LIN {X 0,Y 523.166,Z 946.333,A -85,B 0,C 180,E1 4773.992,E2 4773.992} C_VEL
LIN {X 0,Y 523.378,Z 938.631,A -85,B 0,C 180,E1 4777.898,E2 4777.898} C_VEL
LIN {X 0,Y 523.631,Z 926.038,A -85,B 0,C 180,E1 4781.677,E2 4781.677} C_VEL
LIN {X 0,Y 524.432,Z 907.467,A -85,B 0,C 180,E1 4785.488,E2 4785.488} C_VEL
LIN {X 0,Y 525.679,Z 882.892,A -85,B 0,C 180,E1 4789.124,E2 4789.124} C_VEL
LIN {X 0,Y 527.329,Z 854.452,A -85,B 0,C 180,E1 4792.218,E2 4792.218} C_VEL
LIN {X 0,Y 529.181,Z 823.204,A -85,B 0,C 180,E1 4794.735,E2 4794.735} C_VEL
LIN {X 0,Y 530.972,Z 787.135,A -85,B 0,C 180,E1 4796.792,E2 4796.792} C_VEL
LIN {X 0,Y 531.56,Z 762.454,A -85,B 0,C 180,E1 4797.793,E2 4797.793} C_VEL
LIN {X 0,Y 523.434,Z 741.053,A -85,B 0,C 180,E1 4799.156,E2 4799.156} C_VEL
LIN {X 0,Y 522.497,Z 737.44,A -85,B 0,C 180,E1 4799.385,E2 4799.385} C_VEL
LIN {X 0,Y 522.307,Z 737.44,A -85,B 0,C 180,E1 4805.432,E2 4805.432} C_VEL
LIN {X 0,Y 522.273,Z 737.44,A -85,B 0,C 180,E1 4811.816,E2 4811.816} C_VEL
LIN {X 0,Y 522.371,Z 737.44,A -85,B 0,C 180,E1 4818.204,E2 4818.204} C_VEL
LIN {X 0,Y 522.262,Z 737.44,A -85,B 0,C 180,E1 4824.573,E2 4824.573} C_VEL
LIN {X 0,Y 522.341,Z 737.44,A -85,B 0,C 180,E1 4830.487,E2 4830.487} C_VEL
LIN {X 0,Y 522.548,Z 737.44,A -85,B 0,C 180,E1 4836.077,E2 4836.077} C_VEL
LIN {X 0,Y 522.679,Z 737.44,A -85,B 0,C 180,E1 4841.426,E2 4841.426} C_VEL
LIN {X 0,Y 522.807,Z 737.44,A -85,B 0,C 180,E1 4846.61,E2 4846.61} C_VEL
LIN {X 0,Y 522.85,Z 737.44,A -85,B 0,C 180,E1 4851.68,E2 4851.68} C_VEL
LIN {X 0,Y 522.983,Z 737.44,A -85,B 0,C 180,E1 4856.685,E2 4856.685} C_VEL
LIN {X 0,Y 523.046,Z 737.44,A -85,B 0,C 180,E1 4861.663,E2 4861.663} C_VEL
LIN {X 0,Y 522.917,Z 737.44,A -85,B 0,C 180,E1 4866.654,E2 4866.654} C_VEL
LIN {X 0,Y 522.72,Z 737.44,A -85,B 0,C 180,E1 4871.701,E2 4871.701} C_VEL
LIN {X 0,Y 522.554,Z 737.44,A -85,B 0,C 180,E1 4877.039,E2 4877.039} C_VEL
LIN {X 0,Y 522.579,Z 737.44,A -85,B 0,C 180,E1 4882.128,E2 4882.128} C_VEL
LIN {X 0,Y 522.437,Z 737.44,A -85,B 0,C 180,E1 4887.627,E2 4887.627} C_VEL
LIN {X 0,Y 522.3,Z 737.44,A -85,B 0,C 180,E1 4892.5,E2 4892.5} C_VEL
LIN {X 0,Y 519.848,Z 737.44,A -85,B 0,C 180,E1 4893.914,E2 4893.914} C_VEL
LIN {X 0,Y 514.362,Z 737.44,A -85,B 0,C 180,E1 4896.278,E2 4896.278} C_VEL
LIN {X 0,Y 514.448,Z 737.44,A -85,B 0,C 180,E1 4900.351,E2 4900.351} C_VEL
LIN {X 0,Y 514.369,Z 737.44,A -85,B 0,C 180,E1 4905.056,E2 4905.056} C_VEL
LIN {X 0,Y 514.451,Z 738.219,A -85,B 0,C 180,E1 4908.773,E2 4908.773} C_VEL
LIN {X 0,Y 522.159,Z 752.872,A -85,B 0,C 180,E1 4909.551,E2 4909.551} C_VEL
LIN {X 0,Y 533.735,Z 774.419,A -85,B 0,C 180,E1 4910.952,E2 4910.952} C_VEL
LIN {X 0,Y 532.764,Z 835.83,A -85,B 0,C 180,E1 4912.111,E2 4912.111} C_VEL
LIN {X 0,Y 530.712,Z 877.373,A -85,B 0,C 180,E1 4913.563,E2 4913.563} C_VEL
LIN {X 0,Y 527.965,Z 915.757,A -85,B 0,C 180,E1 4915.56,E2 4915.56} C_VEL
LIN {X 0,Y 524.956,Z 952.662,A -85,B 0,C 180,E1 4918.186,E2 4918.186} C_VEL
LIN {X 0,Y 521.949,Z 987.101,A -85,B 0,C 180,E1 4921.405,E2 4921.405} C_VEL
LIN {X 0,Y 519.457,Z 1016.798,A -85,B 0,C 180,E1 4924.974,E2 4924.974} C_VEL
LIN {X 0,Y 517.473,Z 1044.169,A -85,B 0,C 180,E1 4929.222,E2 4929.222} C_VEL
LIN {X 0,Y 516.306,Z 1064.719,A -85,B 0,C 180,E1 4933.387,E2 4933.387} C_VEL
LIN {X 0,Y 515.508,Z 1081.773,A -85,B 0,C 180,E1 4938.136,E2 4938.136} C_VEL
LIN {X 0,Y 515.302,Z 1091.918,A -85,B 0,C 180,E1 4942.402,E2 4942.402} C_VEL
LIN {X 0,Y 515.21,Z 1097.627,A -85,B 0,C 180,E1 4946.631,E2 4946.631} C_VEL
LIN {X 0,Y 515.166,Z 1099,A -85,B 0,C 180,E1 4950,E2 4950} C_VEL
LIN {X 0,Y 515.206,Z 1097.628,A -85,B 0,C 180,E1 4953.369,E2 4953.369} C_VEL
LIN {X 0,Y 515.35,Z 1091.918,A -85,B 0,C 180,E1 4957.597,E2 4957.597} C_VEL
LIN {X 0,Y 515.5,Z 1081.775,A -85,B 0,C 180,E1 4961.864,E2 4961.864} C_VEL
LIN {X 0,Y 516.118,Z 1066.495,A -85,B 0,C 180,E1 4966.181,E2 4966.181} C_VEL
LIN {X 0,Y 517.333,Z 1045.386,A -85,B 0,C 180,E1 4970.56,E2 4970.56} C_VEL
LIN {X 0,Y 519.164,Z 1019.846,A -85,B 0,C 180,E1 4974.604,E2 4974.604} C_VEL
LIN {X 0,Y 521.782,Z 989.204,A -85,B 0,C 180,E1 4978.368,E2 4978.368} C_VEL
LIN {X 0,Y 524.709,Z 955.261,A -85,B 0,C 180,E1 4981.604,E2 4981.604} C_VEL
LIN {X 0,Y 527.867,Z 917.562,A -85,B 0,C 180,E1 4984.328,E2 4984.328} C_VEL
LIN {X 0,Y 530.645,Z 879.156,A -85,B 0,C 180,E1 4986.358,E2 4986.358} C_VEL
LIN {X 0,Y 532.759,Z 837.651,A -85,B 0,C 180,E1 4987.83,E2 4987.83} C_VEL
LIN {X 0,Y 533.918,Z 785.197,A -85,B 0,C 180,E1 4988.849,E2 4988.849} C_VEL
LIN {X 0,Y 533.297,Z 773.528,A -85,B 0,C 180,E1 4989.101,E2 4989.101} C_VEL
LIN {X 0,Y 515.632,Z 741.65,A -85,B 0,C 180,E1 4991.091,E2 4991.091} C_VEL
LIN {X 0,Y 514.405,Z 737.44,A -85,B 0,C 180,E1 4991.277,E2 4991.277} C_VEL
LIN {X 0,Y 514.421,Z 737.44,A -85,B 0,C 180,E1 4997.396,E2 4997.396} C_VEL
LIN {X 0,Y 514.375,Z 737.44,A -85,B 0,C 180,E1 5002.627,E2 5002.627} C_VEL
LIN {X 0,Y 514.427,Z 737.44,A -85,B 0,C 180,E1 5008.593,E2 5008.593} C_VEL
LIN {X 0,Y 514.57,Z 737.44,A -85,B 0,C 180,E1 5013.808,E2 5013.808} C_VEL
LIN {X 0,Y 514.7,Z 737.44,A -85,B 0,C 180,E1 5020.267,E2 5020.267} C_VEL
LIN {X 0,Y 514.536,Z 737.44,A -85,B 0,C 180,E1 5026.168,E2 5026.168} C_VEL
LIN {X 0,Y 514.81,Z 737.44,A -85,B 0,C 180,E1 5031.541,E2 5031.541} C_VEL
LIN {X 0,Y 514.936,Z 737.44,A -85,B 0,C 180,E1 5036.625,E2 5036.625} C_VEL
LIN {X 0,Y 514.939,Z 737.44,A -85,B 0,C 180,E1 5041.68,E2 5041.68} C_VEL
LIN {X 0,Y 514.889,Z 737.44,A -85,B 0,C 180,E1 5046.75,E2 5046.75} C_VEL
LIN {X 0,Y 514.767,Z 737.44,A -85,B 0,C 180,E1 5051.875,E2 5051.875} C_VEL
LIN {X 0,Y 514.697,Z 737.44,A -85,B 0,C 180,E1 5057.101,E2 5057.101} C_VEL
LIN {X 0,Y 514.616,Z 737.44,A -85,B 0,C 180,E1 5062.479,E2 5062.479} C_VEL
LIN {X 0,Y 514.462,Z 737.44,A -85,B 0,C 180,E1 5068.082,E2 5068.082} C_VEL
LIN {X 0,Y 514.395,Z 737.44,A -85,B 0,C 180,E1 5073.993,E2 5073.993} C_VEL
LIN {X 0,Y 514.349,Z 737.44,A -85,B 0,C 180,E1 5080.349,E2 5080.349} C_VEL
LIN {X 0,Y 514.405,Z 737.44,A -85,B 0,C 180,E1 5085.06,E2 5085.06} C_VEL
LIN {X 0,Y 514.451,Z 737.44,A -85,B 0,C 180,E1 5089.909,E2 5089.909} C_VEL
LIN {X 0,Y 514.344,Z 737.44,A -85,B 0,C 180,E1 5095.995,E2 5095.995} C_VEL
LIN {X 0,Y 514.356,Z 737.853,A -85,B 0,C 180,E1 5099.839,E2 5099.839} C_VEL
LIN {X 0,Y 523.372,Z 760.385,A -85,B 0,C 180,E1 5101.367,E2 5101.367} C_VEL
LIN {X 0,Y 525.202,Z 769.331,A -85,B 0,C 180,E1 5101.888,E2 5101.888} C_VEL
LIN {X 0,Y 523.014,Z 804.439,A -85,B 0,C 180,E1 5103.621,E2 5103.621} C_VEL
LIN {X 0,Y 520.977,Z 837.566,A -85,B 0,C 180,E1 5105.879,E2 5105.879} C_VEL
LIN {X 0,Y 518.918,Z 868.893,A -85,B 0,C 180,E1 5108.828,E2 5108.828} C_VEL
LIN {X 0,Y 517.233,Z 895.151,A -85,B 0,C 180,E1 5112.188,E2 5112.188} C_VEL
LIN {X 0,Y 516.175,Z 916.482,A -85,B 0,C 180,E1 5115.889,E2 5115.889} C_VEL
LIN {X 0,Y 515.578,Z 932.641,A -85,B 0,C 180,E1 5119.852,E2 5119.852} C_VEL
LIN {X 0,Y 515.345,Z 941.867,A -85,B 0,C 180,E1 5123.252,E2 5123.252} C_VEL
LIN {X 0,Y 515.228,Z 947.932,A -85,B 0,C 180,E1 5127.345,E2 5127.345} C_VEL
LIN {X 0,Y 515.27,Z 948.997,A -85,B 0,C 180,E1 5130,E2 5130} C_VEL
LIN {X 0,Y 515.281,Z 946.109,A -85,B 0,C 180,E1 5134.213,E2 5134.213} C_VEL
LIN {X 0,Y 515.507,Z 937.486,A -85,B 0,C 180,E1 5138.444,E2 5138.444} C_VEL
LIN {X 0,Y 515.887,Z 924.305,A -85,B 0,C 180,E1 5142.285,E2 5142.285} C_VEL
LIN {X 0,Y 516.782,Z 905.02,A -85,B 0,C 180,E1 5146.16,E2 5146.16} C_VEL
LIN {X 0,Y 518.157,Z 881.147,A -85,B 0,C 180,E1 5149.634,E2 5149.634} C_VEL
LIN {X 0,Y 519.898,Z 853.939,A -85,B 0,C 180,E1 5152.604,E2 5152.604} C_VEL
LIN {X 0,Y 522.023,Z 821.677,A -85,B 0,C 180,E1 5155.212,E2 5155.212} C_VEL
LIN {X 0,Y 524.446,Z 782.487,A -85,B 0,C 180,E1 5157.458,E2 5157.458} C_VEL
LIN {X 0,Y 524.782,Z 764.25,A -85,B 0,C 180,E1 5158.264,E2 5158.264} C_VEL
LIN {X 0,Y 516.75,Z 742.879,A -85,B 0,C 180,E1 5159.711,E2 5159.711} C_VEL
LIN {X 0,Y 514.477,Z 737.44,A -85,B 0,C 180,E1 5160.14,E2 5160.14} C_VEL
LIN {X 0,Y 514.374,Z 737.44,A -85,B 0,C 180,E1 5166.063,E2 5166.063} C_VEL
LIN {X 0,Y 514.361,Z 737.44,A -85,B 0,C 180,E1 5172.632,E2 5172.632} C_VEL
LIN {X 0,Y 514.44,Z 737.44,A -85,B 0,C 180,E1 5177.409,E2 5177.409} C_VEL
LIN {X 0,Y 514.388,Z 737.44,A -85,B 0,C 180,E1 5182.626,E2 5182.626} C_VEL
LIN {X 0,Y 514.391,Z 737.44,A -85,B 0,C 180,E1 5188.6,E2 5188.6} C_VEL
LIN {X 0,Y 514.568,Z 737.44,A -85,B 0,C 180,E1 5193.818,E2 5193.818} C_VEL
LIN {X 0,Y 514.745,Z 737.44,A -85,B 0,C 180,E1 5200.254,E2 5200.254} C_VEL
LIN {X 0,Y 514.878,Z 737.44,A -85,B 0,C 180,E1 5206.4,E2 5206.4} C_VEL
LIN {X 0,Y 514.96,Z 737.44,A -85,B 0,C 180,E1 5211.552,E2 5211.552} C_VEL
LIN {X 0,Y 515.072,Z 737.44,A -85,B 0,C 180,E1 5216.634,E2 5216.634} C_VEL
LIN {X 0,Y 515.079,Z 737.44,A -85,B 0,C 180,E1 5222.025,E2 5222.025} C_VEL
LIN {X 0,Y 515.005,Z 737.44,A -85,B 0,C 180,E1 5226.757,E2 5226.757} C_VEL
LIN {X 0,Y 514.79,Z 737.44,A -85,B 0,C 180,E1 5231.884,E2 5231.884} C_VEL
LIN {X 0,Y 514.657,Z 737.44,A -85,B 0,C 180,E1 5237.111,E2 5237.111} C_VEL
LIN {X 0,Y 514.634,Z 737.44,A -85,B 0,C 180,E1 5242.488,E2 5242.488} C_VEL
LIN {X 0,Y 514.487,Z 737.44,A -85,B 0,C 180,E1 5248.091,E2 5248.091} C_VEL
LIN {X 0,Y 514.35,Z 737.44,A -85,B 0,C 180,E1 5254.007,E2 5254.007} C_VEL
LIN {X 0,Y 514.362,Z 737.44,A -85,B 0,C 180,E1 5256.278,E2 5256.278} C_VEL
LIN {X 0,Y 513.06,Z 737.44,A -85,B 0,C 180,E1 5257.241,E2 5257.241} C_VEL
LIN {X 0,Y 506.448,Z 737.44,A -85,B 0,C 180,E1 5259.862,E2 5259.862} C_VEL
LIN {X 0,Y 506.359,Z 737.44,A -85,B 0,C 180,E1 5260.111,E2 5260.111} C_VEL
LIN {X 0,Y 506.386,Z 737.44,A -85,B 0,C 180,E1 5265.854,E2 5265.854} C_VEL
LIN {X 0,Y 506.497,Z 737.44,A -85,B 0,C 180,E1 5268.178,E2 5268.178} C_VEL
LIN {X 0,Y 513.949,Z 753.392,A -85,B 0,C 180,E1 5268.981,E2 5268.981} C_VEL
LIN {X 0,Y 527.557,Z 777.284,A -85,B 0,C 180,E1 5270.455,E2 5270.455} C_VEL
LIN {X 0,Y 526.518,Z 835.827,A -85,B 0,C 180,E1 5271.58,E2 5271.58} C_VEL
LIN {X 0,Y 524.251,Z 877.617,A -85,B 0,C 180,E1 5273.051,E2 5273.051} C_VEL
LIN {X 0,Y 521.225,Z 916.8,A -85,B 0,C 180,E1 5275.12,E2 5275.12} C_VEL
LIN {X 0,Y 517.926,Z 953.306,A -85,B 0,C 180,E1 5277.76,E2 5277.76} C_VEL
LIN {X 0,Y 514.769,Z 987.099,A -85,B 0,C 180,E1 5280.969,E2 5280.969} C_VEL
LIN {X 0,Y 511.911,Z 1018.16,A -85,B 0,C 180,E1 5284.777,E2 5284.777} C_VEL
LIN {X 0,Y 509.841,Z 1044.171,A -85,B 0,C 180,E1 5288.896,E2 5288.896} C_VEL
LIN {X 0,Y 508.557,Z 1064.718,A -85,B 0,C 180,E1 5293.126,E2 5293.126} C_VEL
LIN {X 0,Y 507.659,Z 1081.773,A -85,B 0,C 180,E1 5297.95,E2 5297.95} C_VEL
LIN {X 0,Y 507.404,Z 1091.918,A -85,B 0,C 180,E1 5302.283,E2 5302.283} C_VEL
LIN {X 0,Y 507.308,Z 1097.627,A -85,B 0,C 180,E1 5306.578,E2 5306.578} C_VEL
LIN {X 0,Y 507.281,Z 1099,A -85,B 0,C 180,E1 5310,E2 5310} C_VEL
LIN {X 0,Y 507.301,Z 1097.628,A -85,B 0,C 180,E1 5313.422,E2 5313.422} C_VEL
LIN {X 0,Y 507.443,Z 1091.919,A -85,B 0,C 180,E1 5317.716,E2 5317.716} C_VEL
LIN {X 0,Y 507.635,Z 1081.774,A -85,B 0,C 180,E1 5322.05,E2 5322.05} C_VEL
LIN {X 0,Y 508.325,Z 1066.496,A -85,B 0,C 180,E1 5326.436,E2 5326.436} C_VEL
LIN {X 0,Y 509.72,Z 1045.388,A -85,B 0,C 180,E1 5330.881,E2 5330.881} C_VEL
LIN {X 0,Y 511.755,Z 1019.261,A -85,B 0,C 180,E1 5335.07,E2 5335.07} C_VEL
LIN {X 0,Y 514.578,Z 989.203,A -85,B 0,C 180,E1 5338.802,E2 5338.802} C_VEL
LIN {X 0,Y 517.817,Z 954.813,A -85,B 0,C 180,E1 5342.114,E2 5342.114} C_VEL
LIN {X 0,Y 521.131,Z 918.687,A -85,B 0,C 180,E1 5344.76,E2 5344.76} C_VEL
LIN {X 0,Y 524.23,Z 878.854,A -85,B 0,C 180,E1 5346.891,E2 5346.891} C_VEL
LIN {X 0,Y 526.562,Z 837.056,A -85,B 0,C 180,E1 5348.376,E2 5348.376} C_VEL
LIN {X 0,Y 527.773,Z 780.555,A -85,B 0,C 180,E1 5349.469,E2 5349.469} C_VEL
LIN {X 0,Y 526.678,Z 775.495,A -85,B 0,C 180,E1 5349.655,E2 5349.655} C_VEL
LIN {X 0,Y 508.709,Z 743.577,A -85,B 0,C 180,E1 5351.557,E2 5351.557} C_VEL
LIN {X 0,Y 506.504,Z 737.44,A -85,B 0,C 180,E1 5351.882,E2 5351.882} C_VEL
LIN {X 0,Y 506.454,Z 737.44,A -85,B 0,C 180,E1 5358.361,E2 5358.361} C_VEL
LIN {X 0,Y 506.49,Z 737.44,A -85,B 0,C 180,E1 5363.811,E2 5363.811} C_VEL
LIN {X 0,Y 506.5,Z 737.44,A -85,B 0,C 180,E1 5370.094,E2 5370.094} C_VEL
LIN {X 0,Y 506.666,Z 737.44,A -85,B 0,C 180,E1 5375.267,E2 5375.267} C_VEL
LIN {X 0,Y 506.825,Z 737.44,A -85,B 0,C 180,E1 5380.814,E2 5380.814} C_VEL
LIN {X 0,Y 506.65,Z 737.44,A -85,B 0,C 180,E1 5386.166,E2 5386.166} C_VEL
LIN {X 0,Y 506.892,Z 737.44,A -85,B 0,C 180,E1 5391.407,E2 5391.407} C_VEL
LIN {X 0,Y 507.031,Z 737.44,A -85,B 0,C 180,E1 5396.572,E2 5396.572} C_VEL
LIN {X 0,Y 507.039,Z 737.44,A -85,B 0,C 180,E1 5401.706,E2 5401.706} C_VEL
LIN {X 0,Y 506.979,Z 737.44,A -85,B 0,C 180,E1 5406.855,E2 5406.855} C_VEL
LIN {X 0,Y 506.845,Z 737.44,A -85,B 0,C 180,E1 5412.064,E2 5412.064} C_VEL
LIN {X 0,Y 506.775,Z 737.44,A -85,B 0,C 180,E1 5417.376,E2 5417.376} C_VEL
LIN {X 0,Y 506.695,Z 737.44,A -85,B 0,C 180,E1 5422.85,E2 5422.85} C_VEL
LIN {X 0,Y 506.5,Z 737.44,A -85,B 0,C 180,E1 5428.564,E2 5428.564} C_VEL
LIN {X 0,Y 506.472,Z 737.44,A -85,B 0,C 180,E1 5434.6,E2 5434.6} C_VEL
LIN {X 0,Y 506.366,Z 737.44,A -85,B 0,C 180,E1 5441.121,E2 5441.121} C_VEL
LIN {X 0,Y 506.454,Z 737.44,A -85,B 0,C 180,E1 5446.563,E2 5446.563} C_VEL
LIN {X 0,Y 506.475,Z 737.44,A -85,B 0,C 180,E1 5453.284,E2 5453.284} C_VEL
LIN {X 0,Y 506.467,Z 737.589,A -85,B 0,C 180,E1 5459.073,E2 5459.073} C_VEL
LIN {X 0,Y 510.942,Z 747.555,A -85,B 0,C 180,E1 5459.778,E2 5459.778} C_VEL
LIN {X 0,Y 517.56,Z 764.656,A -85,B 0,C 180,E1 5461.014,E2 5461.014} C_VEL
LIN {X 0,Y 518.735,Z 773.411,A -85,B 0,C 180,E1 5461.501,E2 5461.501} C_VEL
LIN {X 0,Y 516.582,Z 805.176,A -85,B 0,C 180,E1 5463.115,E2 5463.115} C_VEL
LIN {X 0,Y 513.935,Z 835.367,A -85,B 0,C 180,E1 5465.295,E2 5465.295} C_VEL
LIN {X 0,Y 511.374,Z 869.182,A -85,B 0,C 180,E1 5468.535,E2 5468.535} C_VEL
LIN {X 0,Y 509.582,Z 895.145,A -85,B 0,C 180,E1 5471.912,E2 5471.912} C_VEL
LIN {X 0,Y 508.367,Z 916.884,A -85,B 0,C 180,E1 5475.75,E2 5475.75} C_VEL
LIN {X 0,Y 507.728,Z 932.639,A -85,B 0,C 180,E1 5479.694,E2 5479.694} C_VEL
LIN {X 0,Y 507.453,Z 941.866,A -85,B 0,C 180,E1 5483.146,E2 5483.146} C_VEL
LIN {X 0,Y 507.342,Z 947.212,A -85,B 0,C 180,E1 5486.578,E2 5486.578} C_VEL
LIN {X 0,Y 507.378,Z 948.997,A -85,B 0,C 180,E1 5490,E2 5490} C_VEL
LIN {X 0,Y 507.384,Z 946.111,A -85,B 0,C 180,E1 5494.278,E2 5494.278} C_VEL
LIN {X 0,Y 507.618,Z 937.488,A -85,B 0,C 180,E1 5498.576,E2 5498.576} C_VEL
LIN {X 0,Y 508.043,Z 924.308,A -85,B 0,C 180,E1 5502.477,E2 5502.477} C_VEL
LIN {X 0,Y 509.012,Z 905.023,A -85,B 0,C 180,E1 5506.413,E2 5506.413} C_VEL
LIN {X 0,Y 510.547,Z 881.152,A -85,B 0,C 180,E1 5509.939,E2 5509.939} C_VEL
LIN {X 0,Y 512.56,Z 852.585,A -85,B 0,C 180,E1 5513.082,E2 5513.082} C_VEL
LIN {X 0,Y 515.422,Z 818.696,A -85,B 0,C 180,E1 5515.909,E2 5515.909} C_VEL
LIN {X 0,Y 517.936,Z 786.373,A -85,B 0,C 180,E1 5517.826,E2 5517.826} C_VEL
LIN {X 0,Y 518.495,Z 767.008,A -85,B 0,C 180,E1 5518.714,E2 5518.714} C_VEL
LIN {X 0,Y 511.71,Z 748.352,A -85,B 0,C 180,E1 5520.036,E2 5520.036} C_VEL
LIN {X 0,Y 506.639,Z 738.499,A -85,B 0,C 180,E1 5520.799,E2 5520.799} C_VEL
LIN {X 0,Y 506.562,Z 737.44,A -85,B 0,C 180,E1 5520.896,E2 5520.896} C_VEL
LIN {X 0,Y 506.44,Z 737.44,A -85,B 0,C 180,E1 5526.719,E2 5526.719} C_VEL
LIN {X 0,Y 506.401,Z 737.44,A -85,B 0,C 180,E1 5533.443,E2 5533.443} C_VEL
LIN {X 0,Y 506.445,Z 737.44,A -85,B 0,C 180,E1 5538.887,E2 5538.887} C_VEL
LIN {X 0,Y 506.42,Z 737.44,A -85,B 0,C 180,E1 5545.396,E2 5545.396} C_VEL
LIN {X 0,Y 506.496,Z 737.44,A -85,B 0,C 180,E1 5551.436,E2 5551.436} C_VEL
LIN {X 0,Y 506.707,Z 737.44,A -85,B 0,C 180,E1 5557.15,E2 5557.15} C_VEL
LIN {X 0,Y 506.904,Z 737.44,A -85,B 0,C 180,E1 5562.893,E2 5562.893} C_VEL
LIN {X 0,Y 506.918,Z 737.44,A -85,B 0,C 180,E1 5567.938,E2 5567.938} C_VEL
LIN {X 0,Y 506.982,Z 737.44,A -85,B 0,C 180,E1 5573.145,E2 5573.145} C_VEL
LIN {X 0,Y 507.041,Z 737.44,A -85,B 0,C 180,E1 5578.294,E2 5578.294} C_VEL
LIN {X 0,Y 507.033,Z 737.44,A -85,B 0,C 180,E1 5583.428,E2 5583.428} C_VEL
LIN {X 0,Y 506.906,Z 737.44,A -85,B 0,C 180,E1 5588.592,E2 5588.592} C_VEL
LIN {X 0,Y 506.821,Z 737.44,A -85,B 0,C 180,E1 5593.83,E2 5593.83} C_VEL
LIN {X 0,Y 506.7,Z 737.44,A -85,B 0,C 180,E1 5599.191,E2 5599.191} C_VEL
LIN {X 0,Y 506.668,Z 737.44,A -85,B 0,C 180,E1 5604.732,E2 5604.732} C_VEL
LIN {X 0,Y 506.489,Z 737.44,A -85,B 0,C 180,E1 5610.544,E2 5610.544} C_VEL
LIN {X 0,Y 506.473,Z 737.44,A -85,B 0,C 180,E1 5616.719,E2 5616.719} C_VEL
LIN {X 0,Y 506.359,Z 737.44,A -85,B 0,C 180,E1 5620.111,E2 5620.111} C_VEL
LIN {X 0,Y 503.864,Z 737.44,A -85,B 0,C 180,E1 5621.571,E2 5621.571} C_VEL
LIN {X 0,Y 498.587,Z 737.44,A -85,B 0,C 180,E1 5623.761,E2 5623.761} C_VEL
LIN {X 0,Y 498.5,Z 737.44,A -85,B 0,C 180,E1 5624.014,E2 5624.014} C_VEL
LIN {X 0,Y 498.611,Z 737.44,A -85,B 0,C 180,E1 5627.574,E2 5627.574} C_VEL
LIN {X 0,Y 508.319,Z 758.234,A -85,B 0,C 180,E1 5628.658,E2 5628.658} C_VEL
LIN {X 0,Y 521.561,Z 781.726,A -85,B 0,C 180,E1 5629.988,E2 5629.988} C_VEL
LIN {X 0,Y 520.326,Z 835.779,A -85,B 0,C 180,E1 5631.035,E2 5631.035} C_VEL
LIN {X 0,Y 517.807,Z 878.549,A -85,B 0,C 180,E1 5632.558,E2 5632.558} C_VEL
LIN {X 0,Y 514.461,Z 918.701,A -85,B 0,C 180,E1 5634.723,E2 5634.723} C_VEL
LIN {X 0,Y 510.665,Z 957.552,A -85,B 0,C 180,E1 5637.631,E2 5637.631} C_VEL
LIN {X 0,Y 506.956,Z 993.552,A -85,B 0,C 180,E1 5641.231,E2 5641.231} C_VEL
LIN {X 0,Y 503.768,Z 1025.525,A -85,B 0,C 180,E1 5645.45,E2 5645.45} C_VEL
LIN {X 0,Y 501.524,Z 1051.369,A -85,B 0,C 180,E1 5649.928,E2 5649.928} C_VEL
LIN {X 0,Y 500.246,Z 1071.518,A -85,B 0,C 180,E1 5654.596,E2 5654.596} C_VEL
LIN {X 0,Y 499.635,Z 1085.29,A -85,B 0,C 180,E1 5659.083,E2 5659.083} C_VEL
LIN {X 0,Y 499.476,Z 1093.479,A -85,B 0,C 180,E1 5663.036,E2 5663.036} C_VEL
LIN {X 0,Y 499.406,Z 1097.627,A -85,B 0,C 180,E1 5666.524,E2 5666.524} C_VEL
LIN {X 0,Y 499.4,Z 1099,A -85,B 0,C 180,E1 5670,E2 5670} C_VEL
LIN {X 0,Y 499.395,Z 1097.628,A -85,B 0,C 180,E1 5673.476,E2 5673.476} C_VEL
LIN {X 0,Y 499.553,Z 1091.919,A -85,B 0,C 180,E1 5677.838,E2 5677.838} C_VEL
LIN {X 0,Y 499.772,Z 1081.774,A -85,B 0,C 180,E1 5682.243,E2 5682.243} C_VEL
LIN {X 0,Y 500.551,Z 1066.497,A -85,B 0,C 180,E1 5686.699,E2 5686.699} C_VEL
LIN {X 0,Y 502.07,Z 1045.389,A -85,B 0,C 180,E1 5691.214,E2 5691.214} C_VEL
LIN {X 0,Y 504.311,Z 1018.984,A -85,B 0,C 180,E1 5695.507,E2 5695.507} C_VEL
LIN {X 0,Y 507.328,Z 989.675,A -85,B 0,C 180,E1 5699.198,E2 5699.198} C_VEL
LIN {X 0,Y 510.781,Z 956.306,A -85,B 0,C 180,E1 5702.475,E2 5702.475} C_VEL
LIN {X 0,Y 514.484,Z 918.702,A -85,B 0,C 180,E1 5705.275,E2 5705.275} C_VEL
LIN {X 0,Y 517.833,Z 879.033,A -85,B 0,C 180,E1 5707.415,E2 5707.415} C_VEL
LIN {X 0,Y 520.32,Z 837.566,A -85,B 0,C 180,E1 5708.905,E2 5708.905} C_VEL
LIN {X 0,Y 521.655,Z 784.779,A -85,B 0,C 180,E1 5709.95,E2 5709.95} C_VEL
LIN {X 0,Y 520.604,Z 778.711,A -85,B 0,C 180,E1 5710.144,E2 5710.144} C_VEL
LIN {X 0,Y 501.405,Z 744.954,A -85,B 0,C 180,E1 5712.079,E2 5712.079} C_VEL
LIN {X 0,Y 498.583,Z 737.44,A -85,B 0,C 180,E1 5712.484,E2 5712.484} C_VEL
LIN {X 0,Y 498.52,Z 737.44,A -85,B 0,C 180,E1 5718.075,E2 5718.075} C_VEL
LIN {X 0,Y 498.527,Z 737.44,A -85,B 0,C 180,E1 5724.757,E2 5724.757} C_VEL
LIN {X 0,Y 498.579,Z 737.44,A -85,B 0,C 180,E1 5730.929,E2 5730.929} C_VEL
LIN {X 0,Y 498.765,Z 737.44,A -85,B 0,C 180,E1 5736.755,E2 5736.755} C_VEL
LIN {X 0,Y 498.881,Z 737.44,A -85,B 0,C 180,E1 5742.33,E2 5742.33} C_VEL
LIN {X 0,Y 498.808,Z 737.44,A -85,B 0,C 180,E1 5747.73,E2 5747.73} C_VEL
LIN {X 0,Y 499.158,Z 737.44,A -85,B 0,C 180,E1 5753.028,E2 5753.028} C_VEL
LIN {X 0,Y 499.381,Z 737.44,A -85,B 0,C 180,E1 5758.258,E2 5758.258} C_VEL
LIN {X 0,Y 499.273,Z 737.44,A -85,B 0,C 180,E1 5763.472,E2 5763.472} C_VEL
LIN {X 0,Y 499.102,Z 737.44,A -85,B 0,C 180,E1 5768.718,E2 5768.718} C_VEL
LIN {X 0,Y 498.934,Z 737.44,A -85,B 0,C 180,E1 5774.043,E2 5774.043} C_VEL
LIN {X 0,Y 498.8,Z 737.44,A -85,B 0,C 180,E1 5779.792,E2 5779.792} C_VEL
LIN {X 0,Y 498.7,Z 737.44,A -85,B 0,C 180,E1 5785.145,E2 5785.145} C_VEL
LIN {X 0,Y 498.542,Z 737.44,A -85,B 0,C 180,E1 5791.755,E2 5791.755} C_VEL
LIN {X 0,Y 498.427,Z 737.44,A -85,B 0,C 180,E1 5797.837,E2 5797.837} C_VEL
LIN {X 0,Y 498.517,Z 737.44,A -85,B 0,C 180,E1 5804.296,E2 5804.296} C_VEL
LIN {X 0,Y 498.485,Z 737.44,A -85,B 0,C 180,E1 5810.372,E2 5810.372} C_VEL
LIN {X 0,Y 498.521,Z 737.44,A -85,B 0,C 180,E1 5816.862,E2 5816.862} C_VEL
LIN {X 0,Y 498.562,Z 737.44,A -85,B 0,C 180,E1 5818.257,E2 5818.257} C_VEL
LIN {X 0,Y 503.137,Z 747.617,A -85,B 0,C 180,E1 5819.011,E2 5819.011} C_VEL
LIN {X 0,Y 510.321,Z 763.929,A -85,B 0,C 180,E1 5820.297,E2 5820.297} C_VEL
LIN {X 0,Y 512.504,Z 774.93,A -85,B 0,C 180,E1 5820.992,E2 5820.992} C_VEL
LIN {X 0,Y 510.118,Z 807.352,A -85,B 0,C 180,E1 5822.673,E2 5822.673} C_VEL
LIN {X 0,Y 507.149,Z 837.974,A -85,B 0,C 180,E1 5824.942,E2 5824.942} C_VEL
LIN {X 0,Y 504.062,Z 868.129,A -85,B 0,C 180,E1 5828.041,E2 5828.041} C_VEL
LIN {X 0,Y 501.844,Z 896.264,A -85,B 0,C 180,E1 5831.798,E2 5831.798} C_VEL
LIN {X 0,Y 500.507,Z 918.03,A -85,B 0,C 180,E1 5835.769,E2 5835.769} C_VEL
LIN {X 0,Y 499.856,Z 932.637,A -85,B 0,C 180,E1 5839.53,E2 5839.53} C_VEL
LIN {X 0,Y 499.561,Z 941.865,A -85,B 0,C 180,E1 5843.037,E2 5843.037} C_VEL
LIN {X 0,Y 499.471,Z 947.211,A -85,B 0,C 180,E1 5846.525,E2 5846.525} C_VEL
LIN {X 0,Y 499.498,Z 948.997,A -85,B 0,C 180,E1 5850,E2 5850} C_VEL
LIN {X 0,Y 499.501,Z 946.111,A -85,B 0,C 180,E1 5854.346,E2 5854.346} C_VEL
LIN {X 0,Y 499.764,Z 937.49,A -85,B 0,C 180,E1 5858.712,E2 5858.712} C_VEL
LIN {X 0,Y 500.218,Z 924.31,A -85,B 0,C 180,E1 5862.676,E2 5862.676} C_VEL
LIN {X 0,Y 501.28,Z 905.026,A -85,B 0,C 180,E1 5866.674,E2 5866.674} C_VEL
LIN {X 0,Y 502.948,Z 881.157,A -85,B 0,C 180,E1 5870.254,E2 5870.254} C_VEL
LIN {X 0,Y 505.934,Z 849.575,A -85,B 0,C 180,E1 5873.896,E2 5873.896} C_VEL
LIN {X 0,Y 508.912,Z 820.136,A -85,B 0,C 180,E1 5876.384,E2 5876.384} C_VEL
LIN {X 0,Y 511.63,Z 787.99,A -85,B 0,C 180,E1 5878.322,E2 5878.322} C_VEL
LIN {X 0,Y 512.161,Z 769.312,A -85,B 0,C 180,E1 5879.211,E2 5879.211} C_VEL
LIN {X 0,Y 505.862,Z 752.546,A -85,B 0,C 180,E1 5880.469,E2 5880.469} C_VEL
LIN {X 0,Y 498.805,Z 739.066,A -85,B 0,C 180,E1 5881.575,E2 5881.575} C_VEL
LIN {X 0,Y 498.635,Z 737.44,A -85,B 0,C 180,E1 5881.718,E2 5881.718} C_VEL
LIN {X 0,Y 498.425,Z 737.44,A -85,B 0,C 180,E1 5887.85,E2 5887.85} C_VEL
LIN {X 0,Y 498.505,Z 737.44,A -85,B 0,C 180,E1 5894.309,E2 5894.309} C_VEL
LIN {X 0,Y 498.48,Z 737.44,A -85,B 0,C 180,E1 5900.381,E2 5900.381} C_VEL
LIN {X 0,Y 498.484,Z 737.44,A -85,B 0,C 180,E1 5906.868,E2 5906.868} C_VEL
LIN {X 0,Y 498.627,Z 737.44,A -85,B 0,C 180,E1 5912.914,E2 5912.914} C_VEL
LIN {X 0,Y 498.846,Z 737.44,A -85,B 0,C 180,E1 5918.648,E2 5918.648} C_VEL
LIN {X 0,Y 498.986,Z 737.44,A -85,B 0,C 180,E1 5924.159,E2 5924.159} C_VEL
LIN {X 0,Y 499.093,Z 737.44,A -85,B 0,C 180,E1 5929.519,E2 5929.519} C_VEL
LIN {X 0,Y 499.141,Z 737.44,A -85,B 0,C 180,E1 5934.784,E2 5934.784} C_VEL
LIN {X 0,Y 499.255,Z 737.44,A -85,B 0,C 180,E1 5940.005,E2 5940.005} C_VEL
LIN {X 0,Y 499.165,Z 737.44,A -85,B 0,C 180,E1 5945.225,E2 5945.225} C_VEL
LIN {X 0,Y 499.003,Z 737.44,A -85,B 0,C 180,E1 5950.492,E2 5950.492} C_VEL
LIN {X 0,Y 498.86,Z 737.44,A -85,B 0,C 180,E1 5955.855,E2 5955.855} C_VEL
LIN {X 0,Y 498.792,Z 737.44,A -85,B 0,C 180,E1 5961.364,E2 5961.364} C_VEL
LIN {X 0,Y 498.64,Z 737.44,A -85,B 0,C 180,E1 5967.096,E2 5967.096} C_VEL
LIN {X 0,Y 498.502,Z 737.44,A -85,B 0,C 180,E1 5973.141,E2 5973.141} C_VEL
LIN {X 0,Y 498.486,Z 737.44,A -85,B 0,C 180,E1 5979.631,E2 5979.631} C_VEL
LIN {X 0,Y 498.5,Z 737.44,A -85,B 0,C 180,E1 5984.014,E2 5984.014} C_VEL
LIN {X 0,Y 494.524,Z 737.44,A -85,B 0,C 180,E1 5985.297,E2 5985.297} C_VEL
LIN {X 0,Y 490.596,Z 737.44,A -85,B 0,C 180,E1 5986.601,E2 5986.601} C_VEL
LIN {X 0,Y 490.662,Z 738.171,A -85,B 0,C 180,E1 5986.978,E2 5986.978} C_VEL
LIN {X 0,Y 504.962,Z 766.638,A -85,B 0,C 180,E1 5988.553,E2 5988.553} C_VEL
LIN {X 0,Y 514.956,Z 784.586,A -85,B 0,C 180,E1 5989.552,E2 5989.552} C_VEL
LIN {X 0,Y 513.998,Z 837.096,A -85,B 0,C 180,E1 5990.533,E2 5990.533} C_VEL
LIN {X 0,Y 511.554,Z 877.526,A -85,B 0,C 180,E1 5991.969,E2 5991.969} C_VEL
LIN {X 0,Y 507.881,Z 918.693,A -85,B 0,C 180,E1 5994.196,E2 5994.196} C_VEL
LIN {X 0,Y 503.793,Z 957.498,A -85,B 0,C 180,E1 5997.129,E2 5997.129} C_VEL
LIN {X 0,Y 499.776,Z 993.772,A -85,B 0,C 180,E1 6000.805,E2 6000.805} C_VEL
LIN {X 0,Y 496.373,Z 1024.941,A -85,B 0,C 180,E1 6004.963,E2 6004.963} C_VEL
LIN {X 0,Y 493.982,Z 1050.272,A -85,B 0,C 180,E1 6009.377,E2 6009.377} C_VEL
LIN {X 0,Y 492.575,Z 1069.983,A -85,B 0,C 180,E1 6013.941,E2 6013.941} C_VEL
LIN {X 0,Y 491.834,Z 1084.143,A -85,B 0,C 180,E1 6018.458,E2 6018.458} C_VEL
LIN {X 0,Y 491.579,Z 1093.479,A -85,B 0,C 180,E1 6022.923,E2 6022.923} C_VEL
LIN {X 0,Y 491.504,Z 1097.627,A -85,B 0,C 180,E1 6026.468,E2 6026.468} C_VEL
LIN {X 0,Y 491.5,Z 1099,A -85,B 0,C 180,E1 6030,E2 6030} C_VEL
LIN {X 0,Y 491.49,Z 1097.628,A -85,B 0,C 180,E1 6033.532,E2 6033.532} C_VEL
LIN {X 0,Y 491.655,Z 1091.919,A -85,B 0,C 180,E1 6037.965,E2 6037.965} C_VEL
LIN {X 0,Y 491.92,Z 1081.773,A -85,B 0,C 180,E1 6042.441,E2 6042.441} C_VEL
LIN {X 0,Y 492.908,Z 1064.858,A -85,B 0,C 180,E1 6047.391,E2 6047.391} C_VEL
LIN {X 0,Y 494.728,Z 1041.691,A -85,B 0,C 180,E1 6052.253,E2 6052.253} C_VEL
LIN {X 0,Y 497.557,Z 1013.532,A -85,B 0,C 180,E1 6056.688,E2 6056.688} C_VEL
LIN {X 0,Y 501.095,Z 981.672,A -85,B 0,C 180,E1 6060.539,E2 6060.539} C_VEL
LIN {X 0,Y 505.114,Z 945.518,A -85,B 0,C 180,E1 6063.876,E2 6063.876} C_VEL
LIN {X 0,Y 509.08,Z 905.991,A -85,B 0,C 180,E1 6066.584,E2 6066.584} C_VEL
LIN {X 0,Y 512.617,Z 863.483,A -85,B 0,C 180,E1 6068.61,E2 6068.61} C_VEL
LIN {X 0,Y 514.701,Z 824.962,A -85,B 0,C 180,E1 6069.737,E2 6069.737} C_VEL
LIN {X 0,Y 514.432,Z 782.453,A -85,B 0,C 180,E1 6070.517,E2 6070.517} C_VEL
LIN {X 0,Y 495.559,Z 749.173,A -85,B 0,C 180,E1 6072.45,E2 6072.45} C_VEL
LIN {X 0,Y 490.657,Z 737.44,A -85,B 0,C 180,E1 6073.086,E2 6073.086} C_VEL
LIN {X 0,Y 490.561,Z 737.44,A -85,B 0,C 180,E1 6079.599,E2 6079.599} C_VEL
LIN {X 0,Y 490.583,Z 737.44,A -85,B 0,C 180,E1 6086.253,E2 6086.253} C_VEL
LIN {X 0,Y 490.695,Z 737.44,A -85,B 0,C 180,E1 6092.429,E2 6092.429} C_VEL
LIN {X 0,Y 490.87,Z 737.44,A -85,B 0,C 180,E1 6098.274,E2 6098.274} C_VEL
LIN {X 0,Y 490.889,Z 737.44,A -85,B 0,C 180,E1 6103.881,E2 6103.881} C_VEL
LIN {X 0,Y 491.021,Z 737.44,A -85,B 0,C 180,E1 6110.634,E2 6110.634} C_VEL
LIN {X 0,Y 491.222,Z 737.44,A -85,B 0,C 180,E1 6116.462,E2 6116.462} C_VEL
LIN {X 0,Y 491.252,Z 737.44,A -85,B 0,C 180,E1 6121.761,E2 6121.761} C_VEL
LIN {X 0,Y 491.156,Z 737.44,A -85,B 0,C 180,E1 6127.077,E2 6127.077} C_VEL
LIN {X 0,Y 491.013,Z 737.44,A -85,B 0,C 180,E1 6132.459,E2 6132.459} C_VEL
LIN {X 0,Y 490.922,Z 737.44,A -85,B 0,C 180,E1 6137.956,E2 6137.956} C_VEL
LIN {X 0,Y 490.807,Z 737.44,A -85,B 0,C 180,E1 6143.634,E2 6143.634} C_VEL
LIN {X 0,Y 490.603,Z 737.44,A -85,B 0,C 180,E1 6150.223,E2 6150.223} C_VEL
LIN {X 0,Y 490.543,Z 737.44,A -85,B 0,C 180,E1 6155.893,E2 6155.893} C_VEL
LIN {X 0,Y 490.59,Z 737.44,A -85,B 0,C 180,E1 6162.75,E2 6162.75} C_VEL
LIN {X 0,Y 490.634,Z 737.44,A -85,B 0,C 180,E1 6167.769,E2 6167.769} C_VEL
LIN {X 0,Y 490.546,Z 737.44,A -85,B 0,C 180,E1 6174.098,E2 6174.098} C_VEL
LIN {X 0,Y 490.609,Z 737.44,A -85,B 0,C 180,E1 6177.439,E2 6177.439} C_VEL
LIN {X 0,Y 495.098,Z 747.292,A -85,B 0,C 180,E1 6178.17,E2 6178.17} C_VEL
LIN {X 0,Y 504.455,Z 767.587,A -85,B 0,C 180,E1 6179.869,E2 6179.869} C_VEL
LIN {X 0,Y 506.306,Z 777.052,A -85,B 0,C 180,E1 6180.491,E2 6180.491} C_VEL
LIN {X 0,Y 503.681,Z 809.848,A -85,B 0,C 180,E1 6182.232,E2 6182.232} C_VEL
LIN {X 0,Y 500.412,Z 840.69,A -85,B 0,C 180,E1 6184.581,E2 6184.581} C_VEL
LIN {X 0,Y 497.146,Z 869.582,A -85,B 0,C 180,E1 6187.625,E2 6187.625} C_VEL
LIN {X 0,Y 494.337,Z 894.601,A -85,B 0,C 180,E1 6191.222,E2 6191.222} C_VEL
LIN {X 0,Y 492.862,Z 916.201,A -85,B 0,C 180,E1 6195.15,E2 6195.15} C_VEL
LIN {X 0,Y 491.997,Z 932.635,A -85,B 0,C 180,E1 6199.36,E2 6199.36} C_VEL
LIN {X 0,Y 491.671,Z 941.863,A -85,B 0,C 180,E1 6202.925,E2 6202.925} C_VEL
LIN {X 0,Y 491.57,Z 947.21,A -85,B 0,C 180,E1 6206.469,E2 6206.469} C_VEL
LIN {X 0,Y 491.598,Z 948.997,A -85,B 0,C 180,E1 6210,E2 6210} C_VEL
LIN {X 0,Y 491.621,Z 946.112,A -85,B 0,C 180,E1 6214.416,E2 6214.416} C_VEL
LIN {X 0,Y 491.872,Z 937.492,A -85,B 0,C 180,E1 6218.853,E2 6218.853} C_VEL
LIN {X 0,Y 492.393,Z 924.312,A -85,B 0,C 180,E1 6222.881,E2 6222.881} C_VEL
LIN {X 0,Y 493.512,Z 905.029,A -85,B 0,C 180,E1 6226.944,E2 6226.944} C_VEL
LIN {X 0,Y 496.354,Z 875.948,A -85,B 0,C 180,E1 6231.471,E2 6231.471} C_VEL
LIN {X 0,Y 499.539,Z 848.228,A -85,B 0,C 180,E1 6234.622,E2 6234.622} C_VEL
LIN {X 0,Y 502.796,Z 818.54,A -85,B 0,C 180,E1 6237.095,E2 6237.095} C_VEL
LIN {X 0,Y 505.654,Z 786.108,A -85,B 0,C 180,E1 6239.011,E2 6239.011} C_VEL
LIN {X 0,Y 506.208,Z 772.998,A -85,B 0,C 180,E1 6239.629,E2 6239.629} C_VEL
LIN {X 0,Y 500.555,Z 757.483,A -85,B 0,C 180,E1 6240.837,E2 6240.837} C_VEL
LIN {X 0,Y 490.939,Z 739.339,A -85,B 0,C 180,E1 6242.364,E2 6242.364} C_VEL
LIN {X 0,Y 490.684,Z 737.44,A -85,B 0,C 180,E1 6242.521,E2 6242.521} C_VEL
LIN {X 0,Y 490.494,Z 737.44,A -85,B 0,C 180,E1 6248.122,E2 6248.122} C_VEL
LIN {X 0,Y 490.583,Z 737.44,A -85,B 0,C 180,E1 6252.761,E2 6252.761} C_VEL
LIN {X 0,Y 490.637,Z 737.44,A -85,B 0,C 180,E1 6257.781,E2 6257.781} C_VEL
LIN {X 0,Y 490.52,Z 737.44,A -85,B 0,C 180,E1 6264.105,E2 6264.105} C_VEL
LIN {X 0,Y 490.588,Z 737.44,A -85,B 0,C 180,E1 6270.419,E2 6270.419} C_VEL
LIN {X 0,Y 490.824,Z 737.44,A -85,B 0,C 180,E1 6276.367,E2 6276.367} C_VEL
LIN {X 0,Y 490.997,Z 737.44,A -85,B 0,C 180,E1 6282.047,E2 6282.047} C_VEL
LIN {X 0,Y 491.09,Z 737.44,A -85,B 0,C 180,E1 6287.543,E2 6287.543} C_VEL
LIN {X 0,Y 491.164,Z 737.44,A -85,B 0,C 180,E1 6292.923,E2 6292.923} C_VEL
LIN {X 0,Y 491.254,Z 737.44,A -85,B 0,C 180,E1 6298.239,E2 6298.239} C_VEL
LIN {X 0,Y 491.224,Z 737.44,A -85,B 0,C 180,E1 6303.538,E2 6303.538} C_VEL
LIN {X 0,Y 491.054,Z 737.44,A -85,B 0,C 180,E1 6309.388,E2 6309.388} C_VEL
LIN {X 0,Y 490.967,Z 737.44,A -85,B 0,C 180,E1 6314.286,E2 6314.286} C_VEL
LIN {X 0,Y 490.854,Z 737.44,A -85,B 0,C 180,E1 6319.836,E2 6319.836} C_VEL
LIN {X 0,Y 490.771,Z 737.44,A -85,B 0,C 180,E1 6325.59,E2 6325.59} C_VEL
LIN {X 0,Y 490.609,Z 737.44,A -85,B 0,C 180,E1 6331.644,E2 6331.644} C_VEL
LIN {X 0,Y 490.555,Z 737.44,A -85,B 0,C 180,E1 6338.118,E2 6338.118} C_VEL
LIN {X 0,Y 490.536,Z 737.44,A -85,B 0,C 180,E1 6344.016,E2 6344.016} C_VEL
LIN {X 0,Y 490.596,Z 737.44,A -85,B 0,C 180,E1 6346.601,E2 6346.601} C_VEL
LIN {X 0,Y 492.101,Z 740.218,A -85,B 0,C 180,E1 6347.102,E2 6347.102} C_VEL
LIN {X 0,Y 494.637,Z 749.813,A -85,B 0,C 180,E1 6347.496,E2 6347.496} C_VEL
LIN {X 0,Y 496.996,Z 767.013,A -85,B 0,C 180,E1 6347.975,E2 6347.975} C_VEL
LIN {X 0,Y 497.957,Z 769.12,A -85,B 0,C 180,E1 6348.087,E2 6348.087} C_VEL
LIN {X 0,Y 508.222,Z 786.689,A -85,B 0,C 180,E1 6349.118,E2 6349.118} C_VEL
LIN {X 0,Y 507.118,Z 838.063,A -85,B 0,C 180,E1 6350.113,E2 6350.113} C_VEL
LIN {X 0,Y 504.832,Z 880.073,A -85,B 0,C 180,E1 6351.561,E2 6351.561} C_VEL
LIN {X 0,Y 501.474,Z 917.434,A -85,B 0,C 180,E1 6353.577,E2 6353.577} C_VEL
LIN {X 0,Y 497.064,Z 956.239,A -85,B 0,C 180,E1 6356.507,E2 6356.507} C_VEL
LIN {X 0,Y 492.934,Z 990.85,A -85,B 0,C 180,E1 6360.005,E2 6360.005} C_VEL
LIN {X 0,Y 489.252,Z 1022.003,A -85,B 0,C 180,E1 6364.115,E2 6364.115} C_VEL
LIN {X 0,Y 486.589,Z 1048.238,A -85,B 0,C 180,E1 6368.645,E2 6368.645} C_VEL
LIN {X 0,Y 484.971,Z 1068.384,A -85,B 0,C 180,E1 6373.253,E2 6373.253} C_VEL
LIN {X 0,Y 484.063,Z 1082.989,A -85,B 0,C 180,E1 6377.812,E2 6377.812} C_VEL
LIN {X 0,Y 483.7,Z 1093.479,A -85,B 0,C 180,E1 6382.808,E2 6382.808} C_VEL
LIN {X 0,Y 483.608,Z 1097.627,A -85,B 0,C 180,E1 6386.41,E2 6386.41} C_VEL
LIN {X 0,Y 483.63,Z 1099,A -85,B 0,C 180,E1 6390,E2 6390} C_VEL
LIN {X 0,Y 483.595,Z 1097.628,A -85,B 0,C 180,E1 6393.59,E2 6393.59} C_VEL
LIN {X 0,Y 483.776,Z 1091.919,A -85,B 0,C 180,E1 6398.096,E2 6398.096} C_VEL
LIN {X 0,Y 484.063,Z 1081.773,A -85,B 0,C 180,E1 6402.646,E2 6402.646} C_VEL
LIN {X 0,Y 485.15,Z 1064.909,A -85,B 0,C 180,E1 6407.666,E2 6407.666} C_VEL
LIN {X 0,Y 487.206,Z 1041.715,A -85,B 0,C 180,E1 6412.611,E2 6412.611} C_VEL
LIN {X 0,Y 490.136,Z 1014.345,A -85,B 0,C 180,E1 6417.01,E2 6417.01} C_VEL
LIN {X 0,Y 494.064,Z 981.716,A -85,B 0,C 180,E1 6421.017,E2 6421.017} C_VEL
LIN {X 0,Y 498.483,Z 944.625,A -85,B 0,C 180,E1 6424.466,E2 6424.466} C_VEL
LIN {X 0,Y 502.743,Z 904.657,A -85,B 0,C 180,E1 6427.207,E2 6427.207} C_VEL
LIN {X 0,Y 505.701,Z 867.042,A -85,B 0,C 180,E1 6428.955,E2 6428.955} C_VEL
LIN {X 0,Y 507.858,Z 825.651,A -85,B 0,C 180,E1 6430.173,E2 6430.173} C_VEL
LIN {X 0,Y 507.725,Z 785.377,A -85,B 0,C 180,E1 6430.938,E2 6430.938} C_VEL
LIN {X 0,Y 489.894,Z 753.751,A -85,B 0,C 180,E1 6432.809,E2 6432.809} C_VEL
LIN {X 0,Y 482.708,Z 737.44,A -85,B 0,C 180,E1 6433.692,E2 6433.692} C_VEL
LIN {X 0,Y 482.659,Z 737.44,A -85,B 0,C 180,E1 6438.835,E2 6438.835} C_VEL
LIN {X 0,Y 482.587,Z 737.44,A -85,B 0,C 180,E1 6444.655,E2 6444.655} C_VEL
LIN {X 0,Y 482.689,Z 737.44,A -85,B 0,C 180,E1 6449.875,E2 6449.875} C_VEL
LIN {X 0,Y 482.874,Z 737.44,A -85,B 0,C 180,E1 6455.943,E2 6455.943} C_VEL
LIN {X 0,Y 483.024,Z 737.44,A -85,B 0,C 180,E1 6461.73,E2 6461.73} C_VEL
LIN {X 0,Y 482.963,Z 737.44,A -85,B 0,C 180,E1 6467.32,E2 6467.32} C_VEL
LIN {X 0,Y 483.312,Z 737.44,A -85,B 0,C 180,E1 6472.798,E2 6472.798} C_VEL
LIN {X 0,Y 483.563,Z 737.44,A -85,B 0,C 180,E1 6478.201,E2 6478.201} C_VEL
LIN {X 0,Y 483.473,Z 737.44,A -85,B 0,C 180,E1 6483.586,E2 6483.586} C_VEL
LIN {X 0,Y 483.266,Z 737.44,A -85,B 0,C 180,E1 6489.007,E2 6489.007} C_VEL
LIN {X 0,Y 483.073,Z 737.44,A -85,B 0,C 180,E1 6494.514,E2 6494.514} C_VEL
LIN {X 0,Y 482.958,Z 737.44,A -85,B 0,C 180,E1 6500.165,E2 6500.165} C_VEL
LIN {X 0,Y 482.814,Z 737.44,A -85,B 0,C 180,E1 6506.033,E2 6506.033} C_VEL
LIN {X 0,Y 482.695,Z 737.44,A -85,B 0,C 180,E1 6512.214,E2 6512.214} C_VEL
LIN {X 0,Y 482.566,Z 737.44,A -85,B 0,C 180,E1 6518.854,E2 6518.854} C_VEL
LIN {X 0,Y 482.618,Z 737.44,A -85,B 0,C 180,E1 6523.82,E2 6523.82} C_VEL
LIN {X 0,Y 482.661,Z 737.44,A -85,B 0,C 180,E1 6528.823,E2 6528.823} C_VEL
LIN {X 0,Y 482.594,Z 737.44,A -85,B 0,C 180,E1 6534.639,E2 6534.639} C_VEL
LIN {X 0,Y 482.704,Z 737.973,A -85,B 0,C 180,E1 6536.707,E2 6536.707} C_VEL
LIN {X 0,Y 489.848,Z 752.147,A -85,B 0,C 180,E1 6537.774,E2 6537.774} C_VEL
LIN {X 0,Y 498.886,Z 772.166,A -85,B 0,C 180,E1 6539.491,E2 6539.491} C_VEL
LIN {X 0,Y 500.061,Z 780.564,A -85,B 0,C 180,E1 6540.029,E2 6540.029} C_VEL
LIN {X 0,Y 497.084,Z 814.322,A -85,B 0,C 180,E1 6541.897,E2 6541.897} C_VEL
LIN {X 0,Y 493.441,Z 845.917,A -85,B 0,C 180,E1 6544.439,E2 6544.439} C_VEL
LIN {X 0,Y 489.794,Z 874.257,A -85,B 0,C 180,E1 6547.604,E2 6547.604} C_VEL
LIN {X 0,Y 486.899,Z 898.153,A -85,B 0,C 180,E1 6551.218,E2 6551.218} C_VEL
LIN {X 0,Y 484.862,Z 919.014,A -85,B 0,C 180,E1 6555.534,E2 6555.534} C_VEL
LIN {X 0,Y 484.06,Z 934.42,A -85,B 0,C 180,E1 6559.792,E2 6559.792} C_VEL
LIN {X 0,Y 483.777,Z 943.53,A -85,B 0,C 180,E1 6563.712,E2 6563.712} C_VEL
LIN {X 0,Y 483.696,Z 948.536,A -85,B 0,C 180,E1 6568.206,E2 6568.206} C_VEL
LIN {X 0,Y 483.693,Z 948.483,A -85,B 0,C 180,E1 6571.794,E2 6571.794} C_VEL
LIN {X 0,Y 483.86,Z 943.374,A -85,B 0,C 180,E1 6576.287,E2 6576.287} C_VEL
LIN {X 0,Y 484.061,Z 934.155,A -85,B 0,C 180,E1 6580.209,E2 6580.209} C_VEL
LIN {X 0,Y 484.886,Z 918.636,A -85,B 0,C 180,E1 6584.465,E2 6584.465} C_VEL
LIN {X 0,Y 486.991,Z 897.581,A -85,B 0,C 180,E1 6588.789,E2 6588.789} C_VEL
LIN {X 0,Y 490.013,Z 872.912,A -85,B 0,C 180,E1 6592.478,E2 6592.478} C_VEL
LIN {X 0,Y 493.685,Z 843.824,A -85,B 0,C 180,E1 6595.669,E2 6595.669} C_VEL
LIN {X 0,Y 497.241,Z 813.243,A -85,B 0,C 180,E1 6598.076,E2 6598.076} C_VEL
LIN {X 0,Y 500.024,Z 782.181,A -85,B 0,C 180,E1 6599.801,E2 6599.801} C_VEL
LIN {X 0,Y 499.804,Z 774.823,A -85,B 0,C 180,E1 6600.196,E2 6600.196} C_VEL
LIN {X 0,Y 493.843,Z 759.405,A -85,B 0,C 180,E1 6601.477,E2 6601.477} C_VEL
LIN {X 0,Y 482.844,Z 738.536,A -85,B 0,C 180,E1 6603.176,E2 6603.176} C_VEL
LIN {X 0,Y 482.762,Z 737.44,A -85,B 0,C 180,E1 6603.406,E2 6603.406} C_VEL
LIN {X 0,Y 482.562,Z 737.44,A -85,B 0,C 180,E1 6608.865,E2 6608.865} C_VEL
LIN {X 0,Y 482.61,Z 737.44,A -85,B 0,C 180,E1 6613.831,E2 6613.831} C_VEL
LIN {X 0,Y 482.668,Z 737.44,A -85,B 0,C 180,E1 6618.835,E2 6618.835} C_VEL
LIN {X 0,Y 482.566,Z 737.44,A -85,B 0,C 180,E1 6624.659,E2 6624.659} C_VEL
LIN {X 0,Y 482.672,Z 737.44,A -85,B 0,C 180,E1 6629.884,E2 6629.884} C_VEL
LIN {X 0,Y 482.862,Z 737.44,A -85,B 0,C 180,E1 6635.953,E2 6635.953} C_VEL
LIN {X 0,Y 483.06,Z 737.44,A -85,B 0,C 180,E1 6641.741,E2 6641.741} C_VEL
LIN {X 0,Y 483.167,Z 737.44,A -85,B 0,C 180,E1 6647.335,E2 6647.335} C_VEL
LIN {X 0,Y 483.263,Z 737.44,A -85,B 0,C 180,E1 6652.806,E2 6652.806} C_VEL
LIN {X 0,Y 483.368,Z 737.44,A -85,B 0,C 180,E1 6658.21,E2 6658.21} C_VEL
LIN {X 0,Y 483.324,Z 737.44,A -85,B 0,C 180,E1 6663.596,E2 6663.596} C_VEL
LIN {X 0,Y 483.183,Z 737.44,A -85,B 0,C 180,E1 6669.018,E2 6669.018} C_VEL
LIN {X 0,Y 483.047,Z 737.44,A -85,B 0,C 180,E1 6674.525,E2 6674.525} C_VEL
LIN {X 0,Y 482.94,Z 737.44,A -85,B 0,C 180,E1 6680.176,E2 6680.176} C_VEL
LIN {X 0,Y 482.854,Z 737.44,A -85,B 0,C 180,E1 6686.041,E2 6686.041} C_VEL
LIN {X 0,Y 482.646,Z 737.44,A -85,B 0,C 180,E1 6692.229,E2 6692.229} C_VEL
LIN {X 0,Y 482.633,Z 737.44,A -85,B 0,C 180,E1 6698.86,E2 6698.86} C_VEL
LIN {X 0,Y 482.637,Z 737.44,A -85,B 0,C 180,E1 6703.822,E2 6703.822} C_VEL
LIN {X 0,Y 482.684,Z 737.44,A -85,B 0,C 180,E1 6706.303,E2 6706.303} C_VEL
LIN {X 0,Y 497.71,Z 768.683,A -85,B 0,C 180,E1 6708.061,E2 6708.061} C_VEL
LIN {X 0,Y 497.957,Z 769.12,A -85,B 0,C 180,E1 6708.087,E2 6708.087} C_VEL
LIN {X 0,Y 501.461,Z 781.151,A -85,B 0,C 180,E1 6708.541,E2 6708.541} C_VEL
LIN {X 0,Y 501.415,Z 803.618,A -85,B 0,C 180,E1 6708.914,E2 6708.914} C_VEL
LIN {X 0,Y 499.702,Z 849.507,A -85,B 0,C 180,E1 6709.992,E2 6709.992} C_VEL
LIN {X 0,Y 496.803,Z 893.647,A -85,B 0,C 180,E1 6711.767,E2 6711.767} C_VEL
LIN {X 0,Y 493.589,Z 929.903,A -85,B 0,C 180,E1 6713.883,E2 6713.883} C_VEL
LIN {X 0,Y 489.082,Z 965.718,A -85,B 0,C 180,E1 6716.862,E2 6716.862} C_VEL
LIN {X 0,Y 484.724,Z 999.084,A -85,B 0,C 180,E1 6720.518,E2 6720.518} C_VEL
LIN {X 0,Y 481.149,Z 1027.874,A -85,B 0,C 180,E1 6724.613,E2 6724.613} C_VEL
LIN {X 0,Y 478.473,Z 1052.466,A -85,B 0,C 180,E1 6729.157,E2 6729.157} C_VEL
LIN {X 0,Y 476.889,Z 1071.685,A -85,B 0,C 180,E1 6733.872,E2 6733.872} C_VEL
LIN {X 0,Y 476.022,Z 1086.437,A -85,B 0,C 180,E1 6738.999,E2 6738.999} C_VEL
LIN {X 0,Y 475.826,Z 1094.703,A -85,B 0,C 180,E1 6743.606,E2 6743.606} C_VEL
LIN {X 0,Y 475.813,Z 1098.657,A -85,B 0,C 180,E1 6748.176,E2 6748.176} C_VEL
LIN {X 0,Y 475.68,Z 1098.657,A -85,B 0,C 180,E1 6751.824,E2 6751.824} C_VEL
LIN {X 0,Y 475.83,Z 1094.704,A -85,B 0,C 180,E1 6756.394,E2 6756.394} C_VEL
LIN {X 0,Y 476.108,Z 1086.438,A -85,B 0,C 180,E1 6760.999,E2 6760.999} C_VEL
LIN {X 0,Y 476.886,Z 1071.685,A -85,B 0,C 180,E1 6766.128,E2 6766.128} C_VEL
LIN {X 0,Y 478.725,Z 1050.359,A -85,B 0,C 180,E1 6771.293,E2 6771.293} C_VEL
LIN {X 0,Y 481.505,Z 1024.945,A -85,B 0,C 180,E1 6775.866,E2 6775.866} C_VEL
LIN {X 0,Y 485.607,Z 992.844,A -85,B 0,C 180,E1 6780.249,E2 6780.249} C_VEL
LIN {X 0,Y 490.196,Z 957.738,A -85,B 0,C 180,E1 6783.882,E2 6783.882} C_VEL
LIN {X 0,Y 494.4,Z 922.081,A -85,B 0,C 180,E1 6786.647,E2 6786.647} C_VEL
LIN {X 0,Y 497.686,Z 882.366,A -85,B 0,C 180,E1 6788.752,E2 6788.752} C_VEL
LIN {X 0,Y 500.262,Z 840.448,A -85,B 0,C 180,E1 6790.266,E2 6790.266} C_VEL
LIN {X 0,Y 501.683,Z 794.284,A -85,B 0,C 180,E1 6791.227,E2 6791.227} C_VEL
LIN {X 0,Y 500.811,Z 787.831,A -85,B 0,C 180,E1 6791.399,E2 6791.399} C_VEL
LIN {X 0,Y 484.187,Z 758.157,A -85,B 0,C 180,E1 6793.187,E2 6793.187} C_VEL
LIN {X 0,Y 474.707,Z 737.44,A -85,B 0,C 180,E1 6794.402,E2 6794.402} C_VEL
LIN {X 0,Y 474.649,Z 737.44,A -85,B 0,C 180,E1 6800.359,E2 6800.359} C_VEL
LIN {X 0,Y 474.655,Z 737.44,A -85,B 0,C 180,E1 6806.028,E2 6806.028} C_VEL
LIN {X 0,Y 474.781,Z 737.44,A -85,B 0,C 180,E1 6811.421,E2 6811.421} C_VEL
LIN {X 0,Y 475.009,Z 737.44,A -85,B 0,C 180,E1 6817.565,E2 6817.565} C_VEL
LIN {X 0,Y 475.058,Z 737.44,A -85,B 0,C 180,E1 6823.328,E2 6823.328} C_VEL
LIN {X 0,Y 475.156,Z 737.44,A -85,B 0,C 180,E1 6828.975,E2 6828.975} C_VEL
LIN {X 0,Y 475.439,Z 737.44,A -85,B 0,C 180,E1 6834.514,E2 6834.514} C_VEL
LIN {X 0,Y 475.561,Z 737.44,A -85,B 0,C 180,E1 6839.995,E2 6839.995} C_VEL
LIN {X 0,Y 475.406,Z 737.44,A -85,B 0,C 180,E1 6845.477,E2 6845.477} C_VEL
LIN {X 0,Y 475.243,Z 737.44,A -85,B 0,C 180,E1 6851.014,E2 6851.014} C_VEL
LIN {X 0,Y 475.065,Z 737.44,A -85,B 0,C 180,E1 6857.046,E2 6857.046} C_VEL
LIN {X 0,Y 474.979,Z 737.44,A -85,B 0,C 180,E1 6862.481,E2 6862.481} C_VEL
LIN {X 0,Y 474.784,Z 737.44,A -85,B 0,C 180,E1 6868.568,E2 6868.568} C_VEL
LIN {X 0,Y 474.697,Z 737.44,A -85,B 0,C 180,E1 6875.027,E2 6875.027} C_VEL
LIN {X 0,Y 474.591,Z 737.44,A -85,B 0,C 180,E1 6882.05,E2 6882.05} C_VEL
LIN {X 0,Y 474.65,Z 737.44,A -85,B 0,C 180,E1 6887.946,E2 6887.946} C_VEL
LIN {X 0,Y 474.682,Z 737.44,A -85,B 0,C 180,E1 6892.866,E2 6892.866} C_VEL
LIN {X 0,Y 474.738,Z 737.44,A -85,B 0,C 180,E1 6895.861,E2 6895.861} C_VEL
LIN {X 0,Y 479.482,Z 747.822,A -85,B 0,C 180,E1 6896.625,E2 6896.625} C_VEL
LIN {X 0,Y 492.59,Z 773.906,A -85,B 0,C 180,E1 6898.894,E2 6898.894} C_VEL
LIN {X 0,Y 493.934,Z 783.673,A -85,B 0,C 180,E1 6899.537,E2 6899.537} C_VEL
LIN {X 0,Y 490.567,Z 818.488,A -85,B 0,C 180,E1 6901.542,E2 6901.542} C_VEL
LIN {X 0,Y 486.751,Z 848.675,A -85,B 0,C 180,E1 6904.062,E2 6904.062} C_VEL
LIN {X 0,Y 482.926,Z 875.874,A -85,B 0,C 180,E1 6907.172,E2 6907.172} C_VEL
LIN {X 0,Y 479.684,Z 899.887,A -85,B 0,C 180,E1 6910.887,E2 6910.887} C_VEL
LIN {X 0,Y 477.316,Z 920.493,A -85,B 0,C 180,E1 6915.301,E2 6915.301} C_VEL
LIN {X 0,Y 476.184,Z 934.958,A -85,B 0,C 180,E1 6919.791,E2 6919.791} C_VEL
LIN {X 0,Y 475.875,Z 943.528,A -85,B 0,C 180,E1 6923.607,E2 6923.607} C_VEL
LIN {X 0,Y 475.792,Z 948.535,A -85,B 0,C 180,E1 6928.177,E2 6928.177} C_VEL
LIN {X 0,Y 475.789,Z 948.483,A -85,B 0,C 180,E1 6931.824,E2 6931.824} C_VEL
LIN {X 0,Y 475.966,Z 943.375,A -85,B 0,C 180,E1 6936.392,E2 6936.392} C_VEL
LIN {X 0,Y 476.293,Z 932.612,A -85,B 0,C 180,E1 6940.995,E2 6940.995} C_VEL
LIN {X 0,Y 477.785,Z 916.351,A -85,B 0,C 180,E1 6945.625,E2 6945.625} C_VEL
LIN {X 0,Y 480.309,Z 895.415,A -85,B 0,C 180,E1 6949.807,E2 6949.807} C_VEL
LIN {X 0,Y 483.828,Z 869.812,A -85,B 0,C 180,E1 6953.514,E2 6953.514} C_VEL
LIN {X 0,Y 487.65,Z 841.703,A -85,B 0,C 180,E1 6956.506,E2 6956.506} C_VEL
LIN {X 0,Y 491.479,Z 810.095,A -85,B 0,C 180,E1 6958.927,E2 6958.927} C_VEL
LIN {X 0,Y 494.023,Z 778.739,A -85,B 0,C 180,E1 6960.616,E2 6960.616} C_VEL
LIN {X 0,Y 487.902,Z 763.089,A -85,B 0,C 180,E1 6961.952,E2 6961.952} C_VEL
LIN {X 0,Y 474.951,Z 738.983,A -85,B 0,C 180,E1 6963.957,E2 6963.957} C_VEL
LIN {X 0,Y 474.772,Z 737.44,A -85,B 0,C 180,E1 6964.078,E2 6964.078} C_VEL
LIN {X 0,Y 474.568,Z 737.44,A -85,B 0,C 180,E1 6970.047,E2 6970.047} C_VEL
LIN {X 0,Y 474.644,Z 737.44,A -85,B 0,C 180,E1 6975.444,E2 6975.444} C_VEL
LIN {X 0,Y 474.65,Z 737.44,A -85,B 0,C 180,E1 6980.372,E2 6980.372} C_VEL
LIN {X 0,Y 474.664,Z 737.44,A -85,B 0,C 180,E1 6987.173,E2 6987.173} C_VEL
LIN {X 0,Y 474.853,Z 737.44,A -85,B 0,C 180,E1 6993.497,E2 6993.497} C_VEL
LIN {X 0,Y 475.089,Z 737.44,A -85,B 0,C 180,E1 6999.486,E2 6999.486} C_VEL
LIN {X 0,Y 475.252,Z 737.44,A -85,B 0,C 180,E1 7005.241,E2 7005.241} C_VEL
LIN {X 0,Y 475.347,Z 737.44,A -85,B 0,C 180,E1 7011.217,E2 7011.217} C_VEL
LIN {X 0,Y 475.561,Z 737.44,A -85,B 0,C 180,E1 7016.354,E2 7016.354} C_VEL
LIN {X 0,Y 475.656,Z 737.44,A -85,B 0,C 180,E1 7021.829,E2 7021.829} C_VEL
LIN {X 0,Y 475.387,Z 737.44,A -85,B 0,C 180,E1 7027.323,E2 7027.323} C_VEL
LIN {X 0,Y 475.164,Z 737.44,A -85,B 0,C 180,E1 7032.891,E2 7032.891} C_VEL
LIN {X 0,Y 475.024,Z 737.44,A -85,B 0,C 180,E1 7038.589,E2 7038.589} C_VEL
LIN {X 0,Y 474.971,Z 737.44,A -85,B 0,C 180,E1 7044.483,E2 7044.483} C_VEL
LIN {X 0,Y 474.731,Z 737.44,A -85,B 0,C 180,E1 7050.684,E2 7050.684} C_VEL
LIN {X 0,Y 474.704,Z 737.44,A -85,B 0,C 180,E1 7057.301,E2 7057.301} C_VEL
LIN {X 0,Y 474.654,Z 737.44,A -85,B 0,C 180,E1 7062.809,E2 7062.809} C_VEL
LIN {X 0,Y 474.711,Z 737.44,A -85,B 0,C 180,E1 7065.593,E2 7065.593} C_VEL
LIN {X 0,Y 493.331,Z 775.471,A -85,B 0,C 180,E1 7067.847,E2 7067.847} C_VEL
LIN {X 0,Y 501.49,Z 789.06,A -85,B 0,C 180,E1 7068.676,E2 7068.676} C_VEL
LIN {X 0,Y 501.415,Z 803.618,A -85,B 0,C 180,E1 7068.914,E2 7068.914} C_VEL
LIN {X 0,Y 497.516,Z 820.737,A -85,B 0,C 180,E1 7068.997,E2 7068.997} C_VEL
LIN {X 0,Y 493.596,Z 835.565,A -85,B 0,C 180,E1 7069.131,E2 7069.131} C_VEL
LIN {X 0,Y 493.452,Z 837.699,A -85,B 0,C 180,E1 7069.19,E2 7069.19} C_VEL
LIN {X 0,Y 490.91,Z 878.839,A -85,B 0,C 180,E1 7070.654,E2 7070.654} C_VEL
LIN {X 0,Y 487.303,Z 920.732,A -85,B 0,C 180,E1 7072.868,E2 7072.868} C_VEL
LIN {X 0,Y 483.473,Z 956.686,A -85,B 0,C 180,E1 7075.487,E2 7075.487} C_VEL
LIN {X 0,Y 478.748,Z 990.949,A -85,B 0,C 180,E1 7079.033,E2 7079.033} C_VEL
LIN {X 0,Y 474.613,Z 1021.307,A -85,B 0,C 180,E1 7083.143,E2 7083.143} C_VEL
LIN {X 0,Y 471.483,Z 1047.41,A -85,B 0,C 180,E1 7087.755,E2 7087.755} C_VEL
LIN {X 0,Y 469.539,Z 1067.688,A -85,B 0,C 180,E1 7092.492,E2 7092.492} C_VEL
LIN {X 0,Y 468.366,Z 1082.99,A -85,B 0,C 180,E1 7097.397,E2 7097.397} C_VEL
LIN {X 0,Y 467.936,Z 1093.479,A -85,B 0,C 180,E1 7102.564,E2 7102.564} C_VEL
LIN {X 0,Y 467.818,Z 1097.627,A -85,B 0,C 180,E1 7106.289,E2 7106.289} C_VEL
LIN {X 0,Y 467.847,Z 1099,A -85,B 0,C 180,E1 7110,E2 7110} C_VEL
LIN {X 0,Y 467.803,Z 1097.628,A -85,B 0,C 180,E1 7113.711,E2 7113.711} C_VEL
LIN {X 0,Y 468.012,Z 1091.919,A -85,B 0,C 180,E1 7118.37,E2 7118.37} C_VEL
LIN {X 0,Y 468.376,Z 1081.771,A -85,B 0,C 180,E1 7123.077,E2 7123.077} C_VEL
LIN {X 0,Y 469.633,Z 1065.566,A -85,B 0,C 180,E1 7128.092,E2 7128.092} C_VEL
LIN {X 0,Y 471.866,Z 1043.558,A -85,B 0,C 180,E1 7133.022,E2 7133.022} C_VEL
LIN {X 0,Y 475.349,Z 1015.861,A -85,B 0,C 180,E1 7137.685,E2 7137.685} C_VEL
LIN {X 0,Y 480.059,Z 982.175,A -85,B 0,C 180,E1 7141.974,E2 7141.974} C_VEL
LIN {X 0,Y 484.385,Z 949.208,A -85,B 0,C 180,E1 7145.136,E2 7145.136} C_VEL
LIN {X 0,Y 488.179,Z 911.05,A -85,B 0,C 180,E1 7147.709,E2 7147.709} C_VEL
LIN {X 0,Y 491.619,Z 869.38,A -85,B 0,C 180,E1 7149.737,E2 7149.737} C_VEL
LIN {X 0,Y 494.215,Z 827.627,A -85,B 0,C 180,E1 7151.055,E2 7151.055} C_VEL
LIN {X 0,Y 494.373,Z 791.17,A -85,B 0,C 180,E1 7151.808,E2 7151.808} C_VEL
LIN {X 0,Y 478.177,Z 762.021,A -85,B 0,C 180,E1 7153.588,E2 7153.588} C_VEL
LIN {X 0,Y 466.775,Z 737.44,A -85,B 0,C 180,E1 7155.175,E2 7155.175} C_VEL
LIN {X 0,Y 466.691,Z 737.44,A -85,B 0,C 180,E1 7161.131,E2 7161.131} C_VEL
LIN {X 0,Y 466.73,Z 737.44,A -85,B 0,C 180,E1 7167.5,E2 7167.5} C_VEL
LIN {X 0,Y 466.926,Z 737.44,A -85,B 0,C 180,E1 7173,E2 7173} C_VEL
LIN {X 0,Y 467.113,Z 737.44,A -85,B 0,C 180,E1 7179.109,E2 7179.109} C_VEL
LIN {X 0,Y 467.091,Z 737.44,A -85,B 0,C 180,E1 7184.967,E2 7184.967} C_VEL
LIN {X 0,Y 467.32,Z 737.44,A -85,B 0,C 180,E1 7190.674,E2 7190.674} C_VEL
LIN {X 0,Y 467.509,Z 737.44,A -85,B 0,C 180,E1 7196.282,E2 7196.282} C_VEL
LIN {X 0,Y 467.563,Z 737.44,A -85,B 0,C 180,E1 7201.851,E2 7201.851} C_VEL
LIN {X 0,Y 467.426,Z 737.44,A -85,B 0,C 180,E1 7207.439,E2 7207.439} C_VEL
LIN {X 0,Y 467.214,Z 737.44,A -85,B 0,C 180,E1 7213.557,E2 7213.557} C_VEL
LIN {X 0,Y 467.08,Z 737.44,A -85,B 0,C 180,E1 7219.948,E2 7219.948} C_VEL
LIN {X 0,Y 466.988,Z 737.44,A -85,B 0,C 180,E1 7224.92,E2 7224.92} C_VEL
LIN {X 0,Y 466.785,Z 737.44,A -85,B 0,C 180,E1 7231.253,E2 7231.253} C_VEL
LIN {X 0,Y 466.653,Z 737.44,A -85,B 0,C 180,E1 7238.046,E2 7238.046} C_VEL
LIN {X 0,Y 466.728,Z 737.44,A -85,B 0,C 180,E1 7244.468,E2 7244.468} C_VEL
LIN {X 0,Y 466.712,Z 737.44,A -85,B 0,C 180,E1 7249.55,E2 7249.55} C_VEL
LIN {X 0,Y 466.816,Z 737.755,A -85,B 0,C 180,E1 7255.081,E2 7255.081} C_VEL
LIN {X 0,Y 471.836,Z 748.194,A -85,B 0,C 180,E1 7255.855,E2 7255.855} C_VEL
LIN {X 0,Y 486.824,Z 778.077,A -85,B 0,C 180,E1 7258.497,E2 7258.497} C_VEL
LIN {X 0,Y 487.781,Z 786.795,A -85,B 0,C 180,E1 7259.041,E2 7259.041} C_VEL
LIN {X 0,Y 484.275,Z 821.139,A -85,B 0,C 180,E1 7261.07,E2 7261.07} C_VEL
LIN {X 0,Y 480.117,Z 851.507,A -85,B 0,C 180,E1 7263.676,E2 7263.676} C_VEL
LIN {X 0,Y 476.012,Z 878.245,A -85,B 0,C 180,E1 7266.823,E2 7266.823} C_VEL
LIN {X 0,Y 472.407,Z 902.453,A -85,B 0,C 180,E1 7270.686,E2 7270.686} C_VEL
LIN {X 0,Y 469.772,Z 922.578,A -85,B 0,C 180,E1 7275.168,E2 7275.168} C_VEL
LIN {X 0,Y 468.564,Z 935.946,A -85,B 0,C 180,E1 7279.444,E2 7279.444} C_VEL
LIN {X 0,Y 468.032,Z 944.171,A -85,B 0,C 180,E1 7283.499,E2 7283.499} C_VEL
LIN {X 0,Y 467.893,Z 948.694,A -85,B 0,C 180,E1 7288.146,E2 7288.146} C_VEL
LIN {X 0,Y 467.891,Z 948.648,A -85,B 0,C 180,E1 7291.854,E2 7291.854} C_VEL
LIN {X 0,Y 468.109,Z 944.025,A -85,B 0,C 180,E1 7296.5,E2 7296.5} C_VEL
LIN {X 0,Y 468.68,Z 934.128,A -85,B 0,C 180,E1 7301.176,E2 7301.176} C_VEL
LIN {X 0,Y 470.359,Z 918.101,A -85,B 0,C 180,E1 7305.879,E2 7305.879} C_VEL
LIN {X 0,Y 473.126,Z 897.454,A -85,B 0,C 180,E1 7310.121,E2 7310.121} C_VEL
LIN {X 0,Y 476.971,Z 872.322,A -85,B 0,C 180,E1 7313.872,E2 7313.872} C_VEL
LIN {X 0,Y 481.234,Z 843.476,A -85,B 0,C 180,E1 7317.014,E2 7317.014} C_VEL
LIN {X 0,Y 485.335,Z 811.979,A -85,B 0,C 180,E1 7319.463,E2 7319.463} C_VEL
LIN {X 0,Y 487.941,Z 781.651,A -85,B 0,C 180,E1 7321.116,E2 7321.116} C_VEL
LIN {X 0,Y 480.096,Z 763.439,A -85,B 0,C 180,E1 7322.718,E2 7322.718} C_VEL
LIN {X 0,Y 466.859,Z 738.327,A -85,B 0,C 180,E1 7324.809,E2 7324.809} C_VEL
LIN {X 0,Y 466.772,Z 737.44,A -85,B 0,C 180,E1 7325.195,E2 7325.195} C_VEL
LIN {X 0,Y 466.672,Z 737.44,A -85,B 0,C 180,E1 7331.753,E2 7331.753} C_VEL
LIN {X 0,Y 466.74,Z 737.44,A -85,B 0,C 180,E1 7338.251,E2 7338.251} C_VEL
LIN {X 0,Y 466.69,Z 737.44,A -85,B 0,C 180,E1 7344.281,E2 7344.281} C_VEL
LIN {X 0,Y 466.809,Z 737.44,A -85,B 0,C 180,E1 7350.898,E2 7350.898} C_VEL
LIN {X 0,Y 467.056,Z 737.44,A -85,B 0,C 180,E1 7357.116,E2 7357.116} C_VEL
LIN {X 0,Y 467.283,Z 737.44,A -85,B 0,C 180,E1 7363.053,E2 7363.053} C_VEL
LIN {X 0,Y 467.407,Z 737.44,A -85,B 0,C 180,E1 7368.799,E2 7368.799} C_VEL
LIN {X 0,Y 467.496,Z 737.44,A -85,B 0,C 180,E1 7374.43,E2 7374.43} C_VEL
LIN {X 0,Y 467.694,Z 737.44,A -85,B 0,C 180,E1 7380.005,E2 7380.005} C_VEL
LIN {X 0,Y 467.525,Z 737.44,A -85,B 0,C 180,E1 7385.579,E2 7385.579} C_VEL
LIN {X 0,Y 467.297,Z 737.44,A -85,B 0,C 180,E1 7391.213,E2 7391.213} C_VEL
LIN {X 0,Y 467.132,Z 737.44,A -85,B 0,C 180,E1 7396.963,E2 7396.963} C_VEL
LIN {X 0,Y 467.051,Z 737.44,A -85,B 0,C 180,E1 7402.895,E2 7402.895} C_VEL
LIN {X 0,Y 466.83,Z 737.44,A -85,B 0,C 180,E1 7409.112,E2 7409.112} C_VEL
LIN {X 0,Y 466.718,Z 737.44,A -85,B 0,C 180,E1 7415.808,E2 7415.808} C_VEL
LIN {X 0,Y 466.747,Z 737.44,A -85,B 0,C 180,E1 7421.75,E2 7421.75} C_VEL
LIN {X 0,Y 466.76,Z 737.44,A -85,B 0,C 180,E1 7424.825,E2 7424.825} C_VEL
LIN {X 0,Y 488.415,Z 781.32,A -85,B 0,C 180,E1 7427.575,E2 7427.575} C_VEL
LIN {X 0,Y 494.651,Z 791.716,A -85,B 0,C 180,E1 7428.226,E2 7428.226} C_VEL
LIN {X 0,Y 493.452,Z 837.699,A -85,B 0,C 180,E1 7429.19,E2 7429.19} C_VEL
LIN {X 0,Y 488.889,Z 854.496,A -85,B 0,C 180,E1 7429.473,E2 7429.473} C_VEL
LIN {X 0,Y 484.601,Z 868.986,A -85,B 0,C 180,E1 7429.801,E2 7429.801} C_VEL
LIN {X 0,Y 484.407,Z 871.065,A -85,B 0,C 180,E1 7429.882,E2 7429.882} C_VEL
LIN {X 0,Y 480.732,Z 914.094,A -85,B 0,C 180,E1 7432.058,E2 7432.058} C_VEL
LIN {X 0,Y 476.414,Z 954.514,A -85,B 0,C 180,E1 7434.926,E2 7434.926} C_VEL
LIN {X 0,Y 473.019,Z 982.51,A -85,B 0,C 180,E1 7437.535,E2 7437.535} C_VEL
LIN {X 0,Y 468.15,Z 1015.377,A -85,B 0,C 180,E1 7441.773,E2 7441.773} C_VEL
LIN {X 0,Y 464.386,Z 1042.549,A -85,B 0,C 180,E1 7446.375,E2 7446.375} C_VEL
LIN {X 0,Y 461.958,Z 1065.128,A -85,B 0,C 180,E1 7451.473,E2 7451.473} C_VEL
LIN {X 0,Y 460.622,Z 1081.769,A -85,B 0,C 180,E1 7456.698,E2 7456.698} C_VEL
LIN {X 0,Y 460.12,Z 1092.104,A -85,B 0,C 180,E1 7461.598,E2 7461.598} C_VEL
LIN {X 0,Y 459.914,Z 1097.627,A -85,B 0,C 180,E1 7466.225,E2 7466.225} C_VEL
LIN {X 0,Y 459.947,Z 1099,A -85,B 0,C 180,E1 7470,E2 7470} C_VEL
LIN {X 0,Y 459.897,Z 1097.628,A -85,B 0,C 180,E1 7473.775,E2 7473.775} C_VEL
LIN {X 0,Y 460.127,Z 1092.103,A -85,B 0,C 180,E1 7478.403,E2 7478.403} C_VEL
LIN {X 0,Y 460.545,Z 1081.771,A -85,B 0,C 180,E1 7483.304,E2 7483.304} C_VEL
LIN {X 0,Y 461.943,Z 1065.228,A -85,B 0,C 180,E1 7488.499,E2 7488.499} C_VEL
LIN {X 0,Y 464.422,Z 1042.481,A -85,B 0,C 180,E1 7493.637,E2 7493.637} C_VEL
LIN {X 0,Y 468.412,Z 1013.675,A -85,B 0,C 180,E1 7498.473,E2 7498.473} C_VEL
LIN {X 0,Y 473.177,Z 981.435,A -85,B 0,C 180,E1 7502.578,E2 7502.578} C_VEL
LIN {X 0,Y 477.136,Z 948.558,A -85,B 0,C 180,E1 7505.55,E2 7505.55} C_VEL
LIN {X 0,Y 481.299,Z 907.905,A -85,B 0,C 180,E1 7508.308,E2 7508.308} C_VEL
LIN {X 0,Y 484.986,Z 864.895,A -85,B 0,C 180,E1 7510.357,E2 7510.357} C_VEL
LIN {X 0,Y 487.67,Z 821.968,A -85,B 0,C 180,E1 7511.665,E2 7511.665} C_VEL
LIN {X 0,Y 487.733,Z 794.15,A -85,B 0,C 180,E1 7512.255,E2 7512.255} C_VEL
LIN {X 0,Y 472.369,Z 766.049,A -85,B 0,C 180,E1 7514.014,E2 7514.014} C_VEL
LIN {X 0,Y 458.831,Z 737.44,A -85,B 0,C 180,E1 7516.037,E2 7516.037} C_VEL
LIN {X 0,Y 458.766,Z 737.44,A -85,B 0,C 180,E1 7522.376,E2 7522.376} C_VEL
LIN {X 0,Y 458.832,Z 737.44,A -85,B 0,C 180,E1 7529.083,E2 7529.083} C_VEL
LIN {X 0,Y 459.047,Z 737.44,A -85,B 0,C 180,E1 7534.608,E2 7534.608} C_VEL
LIN {X 0,Y 459.242,Z 737.44,A -85,B 0,C 180,E1 7540.748,E2 7540.748} C_VEL
LIN {X 0,Y 459.2,Z 737.44,A -85,B 0,C 180,E1 7546.652,E2 7546.652} C_VEL
LIN {X 0,Y 459.535,Z 737.44,A -85,B 0,C 180,E1 7552.423,E2 7552.423} C_VEL
LIN {X 0,Y 459.839,Z 737.44,A -85,B 0,C 180,E1 7558.108,E2 7558.108} C_VEL
LIN {X 0,Y 459.758,Z 737.44,A -85,B 0,C 180,E1 7563.771,E2 7563.771} C_VEL
LIN {X 0,Y 459.512,Z 737.44,A -85,B 0,C 180,E1 7569.476,E2 7569.476} C_VEL
LIN {X 0,Y 459.268,Z 737.44,A -85,B 0,C 180,E1 7575.285,E2 7575.285} C_VEL
LIN {X 0,Y 459.124,Z 737.44,A -85,B 0,C 180,E1 7581.261,E2 7581.261} C_VEL
LIN {X 0,Y 458.95,Z 737.44,A -85,B 0,C 180,E1 7587.497,E2 7587.497} C_VEL
LIN {X 0,Y 458.784,Z 737.44,A -85,B 0,C 180,E1 7594.116,E2 7594.116} C_VEL
LIN {X 0,Y 458.756,Z 737.44,A -85,B 0,C 180,E1 7600.62,E2 7600.62} C_VEL
LIN {X 0,Y 458.821,Z 737.44,A -85,B 0,C 180,E1 7606.535,E2 7606.535} C_VEL
LIN {X 0,Y 458.768,Z 737.44,A -85,B 0,C 180,E1 7612.361,E2 7612.361} C_VEL
LIN {X 0,Y 458.827,Z 737.44,A -85,B 0,C 180,E1 7614.192,E2 7614.192} C_VEL
LIN {X 0,Y 461.482,Z 743.334,A -85,B 0,C 180,E1 7614.628,E2 7614.628} C_VEL
LIN {X 0,Y 479.096,Z 777.641,A -85,B 0,C 180,E1 7617.691,E2 7617.691} C_VEL
LIN {X 0,Y 481.65,Z 787.525,A -85,B 0,C 180,E1 7618.455,E2 7618.455} C_VEL
LIN {X 0,Y 478.264,Z 820.864,A -85,B 0,C 180,E1 7620.397,E2 7620.397} C_VEL
LIN {X 0,Y 474.055,Z 850.962,A -85,B 0,C 180,E1 7622.929,E2 7622.929} C_VEL
LIN {X 0,Y 469.4,Z 878.949,A -85,B 0,C 180,E1 7626.224,E2 7626.224} C_VEL
LIN {X 0,Y 465.456,Z 902.639,A -85,B 0,C 180,E1 7630.031,E2 7630.031} C_VEL
LIN {X 0,Y 462.653,Z 922.134,A -85,B 0,C 180,E1 7634.337,E2 7634.337} C_VEL
LIN {X 0,Y 460.948,Z 937.204,A -85,B 0,C 180,E1 7639.162,E2 7639.162} C_VEL
LIN {X 0,Y 460.288,Z 945.583,A -85,B 0,C 180,E1 7643.389,E2 7643.389} C_VEL
LIN {X 0,Y 460.132,Z 950.044,A -85,B 0,C 180,E1 7648.115,E2 7648.115} C_VEL
LIN {X 0,Y 460.13,Z 950.001,A -85,B 0,C 180,E1 7651.886,E2 7651.886} C_VEL
LIN {X 0,Y 460.361,Z 945.442,A -85,B 0,C 180,E1 7656.61,E2 7656.61} C_VEL
LIN {X 0,Y 461.042,Z 935.673,A -85,B 0,C 180,E1 7661.364,E2 7661.364} C_VEL
LIN {X 0,Y 462.946,Z 919.888,A -85,B 0,C 180,E1 7666.14,E2 7666.14} C_VEL
LIN {X 0,Y 465.995,Z 899.541,A -85,B 0,C 180,E1 7670.442,E2 7670.442} C_VEL
LIN {X 0,Y 470.142,Z 874.876,A -85,B 0,C 180,E1 7674.242,E2 7674.242} C_VEL
LIN {X 0,Y 474.687,Z 846.504,A -85,B 0,C 180,E1 7677.418,E2 7677.418} C_VEL
LIN {X 0,Y 478.906,Z 815.345,A -85,B 0,C 180,E1 7679.884,E2 7679.884} C_VEL
LIN {X 0,Y 481.496,Z 783.58,A -85,B 0,C 180,E1 7681.671,E2 7681.671} C_VEL
LIN {X 0,Y 466.829,Z 753.407,A -85,B 0,C 180,E1 7684.426,E2 7684.426} C_VEL
LIN {X 0,Y 458.961,Z 738.759,A -85,B 0,C 180,E1 7685.65,E2 7685.65} C_VEL
LIN {X 0,Y 458.829,Z 737.44,A -85,B 0,C 180,E1 7685.756,E2 7685.756} C_VEL
LIN {X 0,Y 458.748,Z 737.44,A -85,B 0,C 180,E1 7691.304,E2 7691.304} C_VEL
LIN {X 0,Y 458.82,Z 737.44,A -85,B 0,C 180,E1 7696.548,E2 7696.548} C_VEL
LIN {X 0,Y 458.749,Z 737.44,A -85,B 0,C 180,E1 7702.379,E2 7702.379} C_VEL
LIN {X 0,Y 458.816,Z 737.44,A -85,B 0,C 180,E1 7709.086,E2 7709.086} C_VEL
LIN {X 0,Y 459.027,Z 737.44,A -85,B 0,C 180,E1 7714.618,E2 7714.618} C_VEL
LIN {X 0,Y 459.275,Z 737.44,A -85,B 0,C 180,E1 7720.759,E2 7720.759} C_VEL
LIN {X 0,Y 459.43,Z 737.44,A -85,B 0,C 180,E1 7726.669,E2 7726.669} C_VEL
LIN {X 0,Y 459.526,Z 737.44,A -85,B 0,C 180,E1 7732.433,E2 7732.433} C_VEL
LIN {X 0,Y 459.664,Z 737.44,A -85,B 0,C 180,E1 7738.118,E2 7738.118} C_VEL
LIN {X 0,Y 459.603,Z 737.44,A -85,B 0,C 180,E1 7743.782,E2 7743.782} C_VEL
LIN {X 0,Y 459.446,Z 737.44,A -85,B 0,C 180,E1 7749.488,E2 7749.488} C_VEL
LIN {X 0,Y 459.241,Z 737.44,A -85,B 0,C 180,E1 7755.296,E2 7755.296} C_VEL
LIN {X 0,Y 459.128,Z 737.44,A -85,B 0,C 180,E1 7761.271,E2 7761.271} C_VEL
LIN {X 0,Y 458.975,Z 737.44,A -85,B 0,C 180,E1 7767.507,E2 7767.507} C_VEL
LIN {X 0,Y 458.762,Z 737.44,A -85,B 0,C 180,E1 7774.407,E2 7774.407} C_VEL
LIN {X 0,Y 458.841,Z 737.44,A -85,B 0,C 180,E1 7781.296,E2 7781.296} C_VEL
LIN {X 0,Y 458.831,Z 737.79,A -85,B 0,C 180,E1 7784.061,E2 7784.061} C_VEL
LIN {X 0,Y 483.827,Z 787.654,A -85,B 0,C 180,E1 7787.339,E2 7787.339} C_VEL
LIN {X 0,Y 488.063,Z 794.81,A -85,B 0,C 180,E1 7787.785,E2 7787.785} C_VEL
LIN {X 0,Y 486.421,Z 842.016,A -85,B 0,C 180,E1 7788.848,E2 7788.848} C_VEL
LIN {X 0,Y 484.407,Z 871.065,A -85,B 0,C 180,E1 7789.882,E2 7789.882} C_VEL
LIN {X 0,Y 479.751,Z 887.415,A -85,B 0,C 180,E1 7790.397,E2 7790.397} C_VEL
LIN {X 0,Y 474.626,Z 903.397,A -85,B 0,C 180,E1 7791.019,E2 7791.019} C_VEL
LIN {X 0,Y 470.108,Z 945.629,A -85,B 0,C 180,E1 7793.845,E2 7793.845} C_VEL
LIN {X 0,Y 465.49,Z 983.444,A -85,B 0,C 180,E1 7797.276,E2 7797.276} C_VEL
LIN {X 0,Y 461.986,Z 1008.488,A -85,B 0,C 180,E1 7800.297,E2 7800.297} C_VEL
LIN {X 0,Y 457.749,Z 1036.366,A -85,B 0,C 180,E1 7804.794,E2 7804.794} C_VEL
LIN {X 0,Y 454.783,Z 1058.909,A -85,B 0,C 180,E1 7809.553,E2 7809.553} C_VEL
LIN {X 0,Y 453.131,Z 1076.296,A -85,B 0,C 180,E1 7814.497,E2 7814.497} C_VEL
LIN {X 0,Y 452.349,Z 1088.406,A -85,B 0,C 180,E1 7819.392,E2 7819.392} C_VEL
LIN {X 0,Y 452.118,Z 1095.905,A -85,B 0,C 180,E1 7824.234,E2 7824.234} C_VEL
LIN {X 0,Y 452.106,Z 1098.657,A -85,B 0,C 180,E1 7828.081,E2 7828.081} C_VEL
LIN {X 0,Y 451.986,Z 1098.657,A -85,B 0,C 180,E1 7831.919,E2 7831.919} C_VEL
LIN {X 0,Y 452.14,Z 1094.704,A -85,B 0,C 180,E1 7836.73,E2 7836.73} C_VEL
LIN {X 0,Y 452.455,Z 1086.436,A -85,B 0,C 180,E1 7841.582,E2 7841.582} C_VEL
LIN {X 0,Y 453.553,Z 1071.688,A -85,B 0,C 180,E1 7846.982,E2 7846.982} C_VEL
LIN {X 0,Y 455.932,Z 1050.184,A -85,B 0,C 180,E1 7852.45,E2 7852.45} C_VEL
LIN {X 0,Y 459.697,Z 1023.38,A -85,B 0,C 180,E1 7857.457,E2 7857.457} C_VEL
LIN {X 0,Y 463.882,Z 995.963,A -85,B 0,C 180,E1 7861.343,E2 7861.343} C_VEL
LIN {X 0,Y 468.369,Z 960.733,A -85,B 0,C 180,E1 7864.89,E2 7864.89} C_VEL
LIN {X 0,Y 472.595,Z 923.756,A -85,B 0,C 180,E1 7867.724,E2 7867.724} C_VEL
LIN {X 0,Y 476.523,Z 883.859,A -85,B 0,C 180,E1 7869.983,E2 7869.983} C_VEL
LIN {X 0,Y 479.726,Z 841.138,A -85,B 0,C 180,E1 7871.648,E2 7871.648} C_VEL
LIN {X 0,Y 481.335,Z 797.51,A -85,B 0,C 180,E1 7872.677,E2 7872.677} C_VEL
LIN {X 0,Y 467.304,Z 771.513,A -85,B 0,C 180,E1 7874.372,E2 7874.372} C_VEL
LIN {X 0,Y 452.292,Z 741.859,A -85,B 0,C 180,E1 7876.551,E2 7876.551} C_VEL
LIN {X 0,Y 450.92,Z 737.44,A -85,B 0,C 180,E1 7876.914,E2 7876.914} C_VEL
LIN {X 0,Y 450.85,Z 737.44,A -85,B 0,C 180,E1 7883.701,E2 7883.701} C_VEL
LIN {X 0,Y 450.913,Z 737.44,A -85,B 0,C 180,E1 7889.756,E2 7889.756} C_VEL
LIN {X 0,Y 451.146,Z 737.44,A -85,B 0,C 180,E1 7896.249,E2 7896.249} C_VEL
LIN {X 0,Y 451.29,Z 737.44,A -85,B 0,C 180,E1 7902.423,E2 7902.423} C_VEL
LIN {X 0,Y 451.352,Z 737.44,A -85,B 0,C 180,E1 7908.385,E2 7908.385} C_VEL
LIN {X 0,Y 451.722,Z 737.44,A -85,B 0,C 180,E1 7914.225,E2 7914.225} C_VEL
LIN {X 0,Y 451.901,Z 737.44,A -85,B 0,C 180,E1 7919.995,E2 7919.995} C_VEL
LIN {X 0,Y 451.659,Z 737.44,A -85,B 0,C 180,E1 7925.766,E2 7925.766} C_VEL
LIN {X 0,Y 451.45,Z 737.44,A -85,B 0,C 180,E1 7931.602,E2 7931.602} C_VEL
LIN {X 0,Y 451.31,Z 737.44,A -85,B 0,C 180,E1 7937.566,E2 7937.566} C_VEL
LIN {X 0,Y 451.118,Z 737.44,A -85,B 0,C 180,E1 7943.741,E2 7943.741} C_VEL
LIN {X 0,Y 450.93,Z 737.44,A -85,B 0,C 180,E1 7950.231,E2 7950.231} C_VEL
LIN {X 0,Y 450.829,Z 737.44,A -85,B 0,C 180,E1 7957.182,E2 7957.182} C_VEL
LIN {X 0,Y 450.796,Z 737.44,A -85,B 0,C 180,E1 7962.365,E2 7962.365} C_VEL
LIN {X 0,Y 450.846,Z 737.44,A -85,B 0,C 180,E1 7967.808,E2 7967.808} C_VEL
LIN {X 0,Y 450.868,Z 737.948,A -85,B 0,C 180,E1 7973.326,E2 7973.326} C_VEL
LIN {X 0,Y 456.4,Z 748.628,A -85,B 0,C 180,E1 7974.209,E2 7974.209} C_VEL
LIN {X 0,Y 473.014,Z 781.458,A -85,B 0,C 180,E1 7977.265,E2 7977.265} C_VEL
LIN {X 0,Y 475.384,Z 789.335,A -85,B 0,C 180,E1 7977.921,E2 7977.921} C_VEL
LIN {X 0,Y 471.781,Z 823.109,A -85,B 0,C 180,E1 7979.923,E2 7979.923} C_VEL
LIN {X 0,Y 467.39,Z 853.413,A -85,B 0,C 180,E1 7982.51,E2 7982.51} C_VEL
LIN {X 0,Y 462.787,Z 880.202,A -85,B 0,C 180,E1 7985.683,E2 7985.683} C_VEL
LIN {X 0,Y 458.556,Z 903.431,A -85,B 0,C 180,E1 7989.464,E2 7989.464} C_VEL
LIN {X 0,Y 455.224,Z 923.887,A -85,B 0,C 180,E1 7994.075,E2 7994.075} C_VEL
LIN {X 0,Y 453.323,Z 938.629,A -85,B 0,C 180,E1 7998.928,E2 7998.928} C_VEL
LIN {X 0,Y 452.564,Z 947,A -85,B 0,C 180,E1 8003.276,E2 8003.276} C_VEL
LIN {X 0,Y 452.374,Z 951.395,A -85,B 0,C 180,E1 8008.082,E2 8008.082} C_VEL
LIN {X 0,Y 452.372,Z 951.353,A -85,B 0,C 180,E1 8011.918,E2 8011.918} C_VEL
LIN {X 0,Y 452.624,Z 946.865,A -85,B 0,C 180,E1 8016.723,E2 8016.723} C_VEL
LIN {X 0,Y 453.436,Z 937.23,A -85,B 0,C 180,E1 8021.557,E2 8021.557} C_VEL
LIN {X 0,Y 455.554,Z 921.706,A -85,B 0,C 180,E1 8026.409,E2 8026.409} C_VEL
LIN {X 0,Y 458.883,Z 901.667,A -85,B 0,C 180,E1 8030.774,E2 8030.774} C_VEL
LIN {X 0,Y 463.315,Z 877.35,A -85,B 0,C 180,E1 8034.622,E2 8034.622} C_VEL
LIN {X 0,Y 468.036,Z 849.022,A -85,B 0,C 180,E1 8037.841,E2 8037.841} C_VEL
LIN {X 0,Y 472.544,Z 816.995,A -85,B 0,C 180,E1 8040.405,E2 8040.405} C_VEL
LIN {X 0,Y 475.23,Z 786.403,A -85,B 0,C 180,E1 8042.16,E2 8042.16} C_VEL
LIN {X 0,Y 458.696,Z 753.061,A -85,B 0,C 180,E1 8045.311,E2 8045.311} C_VEL
LIN {X 0,Y 450.901,Z 738.425,A -85,B 0,C 180,E1 8046.563,E2 8046.563} C_VEL
LIN {X 0,Y 450.841,Z 737.44,A -85,B 0,C 180,E1 8046.719,E2 8046.719} C_VEL
LIN {X 0,Y 450.788,Z 737.44,A -85,B 0,C 180,E1 8052.377,E2 8052.377} C_VEL
LIN {X 0,Y 450.847,Z 737.44,A -85,B 0,C 180,E1 8057.819,E2 8057.819} C_VEL
LIN {X 0,Y 450.826,Z 737.44,A -85,B 0,C 180,E1 8063.705,E2 8063.705} C_VEL
LIN {X 0,Y 450.895,Z 737.44,A -85,B 0,C 180,E1 8069.766,E2 8069.766} C_VEL
LIN {X 0,Y 451.139,Z 737.44,A -85,B 0,C 180,E1 8076.26,E2 8076.26} C_VEL
LIN {X 0,Y 451.399,Z 737.44,A -85,B 0,C 180,E1 8082.437,E2 8082.437} C_VEL
LIN {X 0,Y 451.546,Z 737.44,A -85,B 0,C 180,E1 8088.4,E2 8088.4} C_VEL
LIN {X 0,Y 451.664,Z 737.44,A -85,B 0,C 180,E1 8094.234,E2 8094.234} C_VEL
LIN {X 0,Y 451.919,Z 737.44,A -85,B 0,C 180,E1 8100.005,E2 8100.005} C_VEL
LIN {X 0,Y 451.723,Z 737.44,A -85,B 0,C 180,E1 8105.775,E2 8105.775} C_VEL
LIN {X 0,Y 451.436,Z 737.44,A -85,B 0,C 180,E1 8111.613,E2 8111.613} C_VEL
LIN {X 0,Y 451.269,Z 737.44,A -85,B 0,C 180,E1 8117.578,E2 8117.578} C_VEL
LIN {X 0,Y 451.146,Z 737.44,A -85,B 0,C 180,E1 8123.751,E2 8123.751} C_VEL
LIN {X 0,Y 450.913,Z 737.44,A -85,B 0,C 180,E1 8130.244,E2 8130.244} C_VEL
LIN {X 0,Y 450.865,Z 737.44,A -85,B 0,C 180,E1 8137.191,E2 8137.191} C_VEL
LIN {X 0,Y 450.926,Z 738.031,A -85,B 0,C 180,E1 8143.216,E2 8143.216} C_VEL
LIN {X 0,Y 470.439,Z 778.459,A -85,B 0,C 180,E1 8146.063,E2 8146.063} C_VEL
LIN {X 0,Y 481.331,Z 797.524,A -85,B 0,C 180,E1 8147.324,E2 8147.324} C_VEL
LIN {X 0,Y 479.396,Z 846.094,A -85,B 0,C 180,E1 8148.504,E2 8148.504} C_VEL
LIN {X 0,Y 476.088,Z 888.857,A -85,B 0,C 180,E1 8150.253,E2 8150.253} C_VEL
LIN {X 0,Y 474.626,Z 903.397,A -85,B 0,C 180,E1 8151.019,E2 8151.019} C_VEL
LIN {X 0,Y 469.279,Z 919.06,A -85,B 0,C 180,E1 8151.754,E2 8151.754} C_VEL
LIN {X 0,Y 464.458,Z 932.37,A -85,B 0,C 180,E1 8152.479,E2 8152.479} C_VEL
LIN {X 0,Y 464.201,Z 934.21,A -85,B 0,C 180,E1 8152.614,E2 8152.614} C_VEL
LIN {X 0,Y 459.488,Z 971.706,A -85,B 0,C 180,E1 8155.778,E2 8155.778} C_VEL
LIN {X 0,Y 454.982,Z 1005.311,A -85,B 0,C 180,E1 8159.505,E2 8159.505} C_VEL
LIN {X 0,Y 451.551,Z 1028.486,A -85,B 0,C 180,E1 8162.932,E2 8162.932} C_VEL
LIN {X 0,Y 448.122,Z 1052.413,A -85,B 0,C 180,E1 8167.661,E2 8167.661} C_VEL
LIN {X 0,Y 445.888,Z 1071.689,A -85,B 0,C 180,E1 8172.716,E2 8172.716} C_VEL
LIN {X 0,Y 444.574,Z 1086.435,A -85,B 0,C 180,E1 8178.21,E2 8178.21} C_VEL
LIN {X 0,Y 444.244,Z 1094.703,A -85,B 0,C 180,E1 8183.149,E2 8183.149} C_VEL
LIN {X 0,Y 444.199,Z 1098.657,A -85,B 0,C 180,E1 8188.047,E2 8188.047} C_VEL
LIN {X 0,Y 444.083,Z 1098.657,A -85,B 0,C 180,E1 8191.954,E2 8191.954} C_VEL
LIN {X 0,Y 444.258,Z 1094.704,A -85,B 0,C 180,E1 8196.85,E2 8196.85} C_VEL
LIN {X 0,Y 444.594,Z 1086.436,A -85,B 0,C 180,E1 8201.79,E2 8201.79} C_VEL
LIN {X 0,Y 445.801,Z 1071.689,A -85,B 0,C 180,E1 8207.287,E2 8207.287} C_VEL
LIN {X 0,Y 448.362,Z 1050.182,A -85,B 0,C 180,E1 8212.85,E2 8212.85} C_VEL
LIN {X 0,Y 452.421,Z 1023.376,A -85,B 0,C 180,E1 8217.937,E2 8217.937} C_VEL
LIN {X 0,Y 455.996,Z 997.936,A -85,B 0,C 180,E1 8221.389,E2 8221.389} C_VEL
LIN {X 0,Y 460.609,Z 963.19,A -85,B 0,C 180,E1 8225.024,E2 8225.024} C_VEL
LIN {X 0,Y 465.239,Z 925.112,A -85,B 0,C 180,E1 8228.032,E2 8228.032} C_VEL
LIN {X 0,Y 469.419,Z 884.68,A -85,B 0,C 180,E1 8230.39,E2 8230.39} C_VEL
LIN {X 0,Y 472.888,Z 841.497,A -85,B 0,C 180,E1 8232.119,E2 8232.119} C_VEL
LIN {X 0,Y 474.629,Z 800.456,A -85,B 0,C 180,E1 8233.139,E2 8233.139} C_VEL
LIN {X 0,Y 461.06,Z 774.226,A -85,B 0,C 180,E1 8234.921,E2 8234.921} C_VEL
LIN {X 0,Y 445.159,Z 742.869,A -85,B 0,C 180,E1 8237.324,E2 8237.324} C_VEL
LIN {X 0,Y 442.966,Z 737.44,A -85,B 0,C 180,E1 8237.747,E2 8237.747} C_VEL
LIN {X 0,Y 442.904,Z 737.44,A -85,B 0,C 180,E1 8244.468,E2 8244.468} C_VEL
LIN {X 0,Y 443.03,Z 737.44,A -85,B 0,C 180,E1 8251.414,E2 8251.414} C_VEL
LIN {X 0,Y 443.262,Z 737.44,A -85,B 0,C 180,E1 8257.928,E2 8257.928} C_VEL
LIN {X 0,Y 443.325,Z 737.44,A -85,B 0,C 180,E1 8264.141,E2 8264.141} C_VEL
LIN {X 0,Y 443.559,Z 737.44,A -85,B 0,C 180,E1 8270.169,E2 8270.169} C_VEL
LIN {X 0,Y 443.786,Z 737.44,A -85,B 0,C 180,E1 8276.083,E2 8276.083} C_VEL
LIN {X 0,Y 443.872,Z 737.44,A -85,B 0,C 180,E1 8281.949,E2 8281.949} C_VEL
LIN {X 0,Y 443.666,Z 737.44,A -85,B 0,C 180,E1 8288.267,E2 8288.267} C_VEL
LIN {X 0,Y 443.459,Z 737.44,A -85,B 0,C 180,E1 8293.82,E2 8293.82} C_VEL
LIN {X 0,Y 443.322,Z 737.44,A -85,B 0,C 180,E1 8299.962,E2 8299.962} C_VEL
LIN {X 0,Y 443.107,Z 737.44,A -85,B 0,C 180,E1 8306.363,E2 8306.363} C_VEL
LIN {X 0,Y 442.941,Z 737.44,A -85,B 0,C 180,E1 8313.144,E2 8313.144} C_VEL
LIN {X 0,Y 442.837,Z 737.44,A -85,B 0,C 180,E1 8318.156,E2 8318.156} C_VEL
LIN {X 0,Y 442.852,Z 737.44,A -85,B 0,C 180,E1 8324.116,E2 8324.116} C_VEL
LIN {X 0,Y 442.857,Z 737.44,A -85,B 0,C 180,E1 8329.493,E2 8329.493} C_VEL
LIN {X 0,Y 442.906,Z 737.44,A -85,B 0,C 180,E1 8332.362,E2 8332.362} C_VEL
LIN {X 0,Y 445.51,Z 743.22,A -85,B 0,C 180,E1 8332.819,E2 8332.819} C_VEL
LIN {X 0,Y 463.324,Z 777.683,A -85,B 0,C 180,E1 8336.06,E2 8336.06} C_VEL
LIN {X 0,Y 469.116,Z 790.802,A -85,B 0,C 180,E1 8337.362,E2 8337.362} C_VEL
LIN {X 0,Y 465.324,Z 824.822,A -85,B 0,C 180,E1 8339.409,E2 8339.409} C_VEL
LIN {X 0,Y 460.861,Z 854.377,A -85,B 0,C 180,E1 8341.954,E2 8341.954} C_VEL
LIN {X 0,Y 455.974,Z 881.784,A -85,B 0,C 180,E1 8345.217,E2 8345.217} C_VEL
LIN {X 0,Y 451.678,Z 904.271,A -85,B 0,C 180,E1 8348.88,E2 8348.88} C_VEL
LIN {X 0,Y 448.071,Z 923.905,A -85,B 0,C 180,E1 8353.309,E2 8353.309} C_VEL
LIN {X 0,Y 445.818,Z 939.014,A -85,B 0,C 180,E1 8358.243,E2 8358.243} C_VEL
LIN {X 0,Y 444.829,Z 948.425,A -85,B 0,C 180,E1 8363.159,E2 8363.159} C_VEL
LIN {X 0,Y 444.612,Z 952.747,A -85,B 0,C 180,E1 8368.049,E2 8368.049} C_VEL
LIN {X 0,Y 444.611,Z 952.706,A -85,B 0,C 180,E1 8371.952,E2 8371.952} C_VEL
LIN {X 0,Y 444.888,Z 948.295,A -85,B 0,C 180,E1 8376.841,E2 8376.841} C_VEL
LIN {X 0,Y 445.826,Z 938.807,A -85,B 0,C 180,E1 8381.757,E2 8381.757} C_VEL
LIN {X 0,Y 448.185,Z 923.549,A -85,B 0,C 180,E1 8386.687,E2 8386.687} C_VEL
LIN {X 0,Y 451.796,Z 903.797,A -85,B 0,C 180,E1 8391.114,E2 8391.114} C_VEL
LIN {X 0,Y 456.097,Z 881.168,A -85,B 0,C 180,E1 8394.777,E2 8394.777} C_VEL
LIN {X 0,Y 460.972,Z 853.564,A -85,B 0,C 180,E1 8398.039,E2 8398.039} C_VEL
LIN {X 0,Y 465.704,Z 822.316,A -85,B 0,C 180,E1 8400.681,E2 8400.681} C_VEL
LIN {X 0,Y 468.823,Z 789.053,A -85,B 0,C 180,E1 8402.678,E2 8402.678} C_VEL
LIN {X 0,Y 451.829,Z 754.747,A -85,B 0,C 180,E1 8406.027,E2 8406.027} C_VEL
LIN {X 0,Y 442.913,Z 738.078,A -85,B 0,C 180,E1 8407.511,E2 8407.511} C_VEL
LIN {X 0,Y 442.847,Z 737.44,A -85,B 0,C 180,E1 8414.127,E2 8414.127} C_VEL
LIN {X 0,Y 442.858,Z 737.44,A -85,B 0,C 180,E1 8419.503,E2 8419.503} C_VEL
LIN {X 0,Y 442.903,Z 737.44,A -85,B 0,C 180,E1 8425.125,E2 8425.125} C_VEL
LIN {X 0,Y 443.01,Z 737.44,A -85,B 0,C 180,E1 8431.424,E2 8431.424} C_VEL
LIN {X 0,Y 443.274,Z 737.44,A -85,B 0,C 180,E1 8437.94,E2 8437.94} C_VEL
LIN {X 0,Y 443.506,Z 737.44,A -85,B 0,C 180,E1 8444.158,E2 8444.158} C_VEL
LIN {X 0,Y 443.703,Z 737.44,A -85,B 0,C 180,E1 8450.183,E2 8450.183} C_VEL
LIN {X 0,Y 443.944,Z 737.44,A -85,B 0,C 180,E1 8456.094,E2 8456.094} C_VEL
LIN {X 0,Y 444.035,Z 737.44,A -85,B 0,C 180,E1 8461.959,E2 8461.959} C_VEL
LIN {X 0,Y 443.66,Z 737.44,A -85,B 0,C 180,E1 8468.26,E2 8468.26} C_VEL
LIN {X 0,Y 443.456,Z 737.44,A -85,B 0,C 180,E1 8473.831,E2 8473.831} C_VEL
LIN {X 0,Y 443.312,Z 737.44,A -85,B 0,C 180,E1 8479.973,E2 8479.973} C_VEL
LIN {X 0,Y 443.136,Z 737.44,A -85,B 0,C 180,E1 8486.372,E2 8486.372} C_VEL
LIN {X 0,Y 442.918,Z 737.44,A -85,B 0,C 180,E1 8493.159,E2 8493.159} C_VEL
LIN {X 0,Y 442.891,Z 737.44,A -85,B 0,C 180,E1 8498.165,E2 8498.165} C_VEL
LIN {X 0,Y 442.979,Z 737.99,A -85,B 0,C 180,E1 8502.314,E2 8502.314} C_VEL
LIN {X 0,Y 462.598,Z 777.559,A -85,B 0,C 180,E1 8505.303,E2 8505.303} C_VEL
LIN {X 0,Y 474.63,Z 800.467,A -85,B 0,C 180,E1 8506.861,E2 8506.861} C_VEL
LIN {X 0,Y 472.527,Z 845.962,A -85,B 0,C 180,E1 8508.024,E2 8508.024} C_VEL
LIN {X 0,Y 469.053,Z 888.435,A -85,B 0,C 180,E1 8509.793,E2 8509.793} C_VEL
LIN {X 0,Y 464.785,Z 929.123,A -85,B 0,C 180,E1 8512.238,E2 8512.238} C_VEL
LIN {X 0,Y 464.201,Z 934.21,A -85,B 0,C 180,E1 8512.614,E2 8512.614} C_VEL
LIN {X 0,Y 460.692,Z 945.475,A -85,B 0,C 180,E1 8513.359,E2 8513.359} C_VEL
LIN {X 0,Y 453.465,Z 961.486,A -85,B 0,C 180,E1 8514.483,E2 8514.483} C_VEL
LIN {X 0,Y 453.092,Z 963.24,A -85,B 0,C 180,E1 8514.637,E2 8514.637} C_VEL
LIN {X 0,Y 448.407,Z 997.674,A -85,B 0,C 180,E1 8518.301,E2 8518.301} C_VEL
LIN {X 0,Y 444.231,Z 1027.327,A -85,B 0,C 180,E1 8522.39,E2 8522.39} C_VEL
LIN {X 0,Y 441.143,Z 1047.779,A -85,B 0,C 180,E1 8526.218,E2 8526.218} C_VEL
LIN {X 0,Y 438.454,Z 1068.661,A -85,B 0,C 180,E1 8531.5,E2 8531.5} C_VEL
LIN {X 0,Y 436.919,Z 1084.14,A -85,B 0,C 180,E1 8536.983,E2 8536.983} C_VEL
LIN {X 0,Y 436.39,Z 1093.479,A -85,B 0,C 180,E1 8542.023,E2 8542.023} C_VEL
LIN {X 0,Y 436.229,Z 1097.627,A -85,B 0,C 180,E1 8546.02,E2 8546.02} C_VEL
LIN {X 0,Y 436.256,Z 1099,A -85,B 0,C 180,E1 8550,E2 8550} C_VEL
LIN {X 0,Y 436.21,Z 1097.628,A -85,B 0,C 180,E1 8553.98,E2 8553.98} C_VEL
LIN {X 0,Y 436.484,Z 1091.833,A -85,B 0,C 180,E1 8559.035,E2 8559.035} C_VEL
LIN {X 0,Y 437.214,Z 1080.567,A -85,B 0,C 180,E1 8564.488,E2 8564.488} C_VEL
LIN {X 0,Y 438.861,Z 1064.703,A -85,B 0,C 180,E1 8569.655,E2 8569.655} C_VEL
LIN {X 0,Y 442.13,Z 1041.869,A -85,B 0,C 180,E1 8575.033,E2 8575.033} C_VEL
LIN {X 0,Y 445.22,Z 1020.212,A -85,B 0,C 180,E1 8578.686,E2 8578.686} C_VEL
LIN {X 0,Y 449.813,Z 987.938,A -85,B 0,C 180,E1 8582.841,E2 8582.841} C_VEL
LIN {X 0,Y 454.81,Z 950.531,A -85,B 0,C 180,E1 8586.486,E2 8586.486} C_VEL
LIN {X 0,Y 459.512,Z 910.832,A -85,B 0,C 180,E1 8589.381,E2 8589.381} C_VEL
LIN {X 0,Y 463.991,Z 867.667,A -85,B 0,C 180,E1 8591.624,E2 8591.624} C_VEL
LIN {X 0,Y 467.483,Z 823.163,A -85,B 0,C 180,E1 8593.142,E2 8593.142} C_VEL
LIN {X 0,Y 467.719,Z 802.875,A -85,B 0,C 180,E1 8593.67,E2 8593.67} C_VEL
LIN {X 0,Y 453.988,Z 774.881,A -85,B 0,C 180,E1 8595.628,E2 8595.628} C_VEL
LIN {X 0,Y 437.392,Z 743.096,A -85,B 0,C 180,E1 8598.232,E2 8598.232} C_VEL
LIN {X 0,Y 434.976,Z 737.44,A -85,B 0,C 180,E1 8598.781,E2 8598.781} C_VEL
LIN {X 0,Y 434.995,Z 737.44,A -85,B 0,C 180,E1 8606.157,E2 8606.157} C_VEL
LIN {X 0,Y 435.185,Z 737.44,A -85,B 0,C 180,E1 8613.107,E2 8613.107} C_VEL
LIN {X 0,Y 435.454,Z 737.44,A -85,B 0,C 180,E1 8619.84,E2 8619.84} C_VEL
LIN {X 0,Y 435.458,Z 737.44,A -85,B 0,C 180,E1 8626.779,E2 8626.779} C_VEL
LIN {X 0,Y 435.79,Z 737.44,A -85,B 0,C 180,E1 8632.007,E2 8632.007} C_VEL
LIN {X 0,Y 436.148,Z 737.44,A -85,B 0,C 180,E1 8638.006,E2 8638.006} C_VEL
LIN {X 0,Y 436.023,Z 737.44,A -85,B 0,C 180,E1 8643.977,E2 8643.977} C_VEL
LIN {X 0,Y 435.723,Z 737.44,A -85,B 0,C 180,E1 8649.999,E2 8649.999} C_VEL
LIN {X 0,Y 435.508,Z 737.44,A -85,B 0,C 180,E1 8656.141,E2 8656.141} C_VEL
LIN {X 0,Y 435.298,Z 737.44,A -85,B 0,C 180,E1 8662.486,E2 8662.486} C_VEL
LIN {X 0,Y 435.038,Z 737.44,A -85,B 0,C 180,E1 8669.149,E2 8669.149} C_VEL
LIN {X 0,Y 435.002,Z 737.44,A -85,B 0,C 180,E1 8673.83,E2 8673.83} C_VEL
LIN {X 0,Y 434.873,Z 737.44,A -85,B 0,C 180,E1 8680.011,E2 8680.011} C_VEL
LIN {X 0,Y 434.968,Z 737.44,A -85,B 0,C 180,E1 8685.882,E2 8685.882} C_VEL
LIN {X 0,Y 434.92,Z 737.44,A -85,B 0,C 180,E1 8691.377,E2 8691.377} C_VEL
LIN {X 0,Y 437.454,Z 743.185,A -85,B 0,C 180,E1 8691.841,E2 8691.841} C_VEL
LIN {X 0,Y 454.005,Z 774.757,A -85,B 0,C 180,E1 8694.909,E2 8694.909} C_VEL
LIN {X 0,Y 462.57,Z 793.057,A -85,B 0,C 180,E1 8696.81,E2 8696.81} C_VEL
LIN {X 0,Y 458.87,Z 826.629,A -85,B 0,C 180,E1 8698.897,E2 8698.897} C_VEL
LIN {X 0,Y 454.14,Z 856.362,A -85,B 0,C 180,E1 8701.501,E2 8701.501} C_VEL
LIN {X 0,Y 449.282,Z 882.264,A -85,B 0,C 180,E1 8704.608,E2 8704.608} C_VEL
LIN {X 0,Y 444.737,Z 904.827,A -85,B 0,C 180,E1 8708.272,E2 8708.272} C_VEL
LIN {X 0,Y 441.044,Z 923.848,A -85,B 0,C 180,E1 8712.521,E2 8712.521} C_VEL
LIN {X 0,Y 438.395,Z 939.438,A -85,B 0,C 180,E1 8717.535,E2 8717.535} C_VEL
LIN {X 0,Y 437.296,Z 948.466,A -85,B 0,C 180,E1 8722.04,E2 8722.04} C_VEL
LIN {X 0,Y 436.863,Z 952.974,A -85,B 0,C 180,E1 8726.026,E2 8726.026} C_VEL
LIN {X 0,Y 436.868,Z 954.491,A -85,B 0,C 180,E1 8730,E2 8730} C_VEL
LIN {X 0,Y 436.874,Z 952.907,A -85,B 0,C 180,E1 8733.975,E2 8733.975} C_VEL
LIN {X 0,Y 437.464,Z 947.049,A -85,B 0,C 180,E1 8738.706,E2 8738.706} C_VEL
LIN {X 0,Y 439.067,Z 935.166,A -85,B 0,C 180,E1 8743.968,E2 8743.968} C_VEL
LIN {X 0,Y 442.101,Z 918.025,A -85,B 0,C 180,E1 8748.85,E2 8748.85} C_VEL
LIN {X 0,Y 446.432,Z 896.383,A -85,B 0,C 180,E1 8753.145,E2 8753.145} C_VEL
LIN {X 0,Y 451.693,Z 869.589,A -85,B 0,C 180,E1 8756.951,E2 8756.951} C_VEL
LIN {X 0,Y 456.944,Z 839.407,A -85,B 0,C 180,E1 8759.999,E2 8759.999} C_VEL
LIN {X 0,Y 461.368,Z 806.309,A -85,B 0,C 180,E1 8762.359,E2 8762.359} C_VEL
LIN {X 0,Y 462.536,Z 792.582,A -85,B 0,C 180,E1 8763.129,E2 8763.129} C_VEL
LIN {X 0,Y 445.676,Z 757.989,A -85,B 0,C 180,E1 8766.64,E2 8766.64} C_VEL
LIN {X 0,Y 435.046,Z 738.888,A -85,B 0,C 180,E1 8768.464,E2 8768.464} C_VEL
LIN {X 0,Y 434.878,Z 737.44,A -85,B 0,C 180,E1 8768.627,E2 8768.627} C_VEL
LIN {X 0,Y 434.946,Z 737.44,A -85,B 0,C 180,E1 8774.121,E2 8774.121} C_VEL
LIN {X 0,Y 434.912,Z 737.44,A -85,B 0,C 180,E1 8779.983,E2 8779.983} C_VEL
LIN {X 0,Y 435,Z 737.44,A -85,B 0,C 180,E1 8786.648,E2 8786.648} C_VEL
LIN {X 0,Y 435.162,Z 737.44,A -85,B 0,C 180,E1 8793.118,E2 8793.118} C_VEL
LIN {X 0,Y 435.476,Z 737.44,A -85,B 0,C 180,E1 8799.833,E2 8799.833} C_VEL
LIN {X 0,Y 435.635,Z 737.44,A -85,B 0,C 180,E1 8806.681,E2 8806.681} C_VEL
LIN {X 0,Y 435.829,Z 737.44,A -85,B 0,C 180,E1 8812.019,E2 8812.019} C_VEL
LIN {X 0,Y 435.989,Z 737.44,A -85,B 0,C 180,E1 8818.015,E2 8818.015} C_VEL
LIN {X 0,Y 435.879,Z 737.44,A -85,B 0,C 180,E1 8823.988,E2 8823.988} C_VEL
LIN {X 0,Y 435.68,Z 737.44,A -85,B 0,C 180,E1 8830.01,E2 8830.01} C_VEL
LIN {X 0,Y 435.457,Z 737.44,A -85,B 0,C 180,E1 8836.153,E2 8836.153} C_VEL
LIN {X 0,Y 435.316,Z 737.44,A -85,B 0,C 180,E1 8842.497,E2 8842.497} C_VEL
LIN {X 0,Y 435.038,Z 737.44,A -85,B 0,C 180,E1 8849.161,E2 8849.161} C_VEL
LIN {X 0,Y 434.997,Z 737.44,A -85,B 0,C 180,E1 8853.843,E2 8853.843} C_VEL
LIN {X 0,Y 434.999,Z 737.44,A -85,B 0,C 180,E1 8861.308,E2 8861.308} C_VEL
LIN {X 0,Y 437.73,Z 743.362,A -85,B 0,C 180,E1 8861.821,E2 8861.821} C_VEL
LIN {X 0,Y 455.287,Z 777.765,A -85,B 0,C 180,E1 8864.573,E2 8864.573} C_VEL
LIN {X 0,Y 468.126,Z 803.547,A -85,B 0,C 180,E1 8866.382,E2 8866.382} C_VEL
LIN {X 0,Y 465.604,Z 847.441,A -85,B 0,C 180,E1 8867.588,E2 8867.588} C_VEL
LIN {X 0,Y 461.825,Z 890.268,A -85,B 0,C 180,E1 8869.452,E2 8869.452} C_VEL
LIN {X 0,Y 457.333,Z 930.682,A -85,B 0,C 180,E1 8871.956,E2 8871.956} C_VEL
LIN {X 0,Y 453.092,Z 963.24,A -85,B 0,C 180,E1 8874.637,E2 8874.637} C_VEL
LIN {X 0,Y 447.495,Z 977.086,A -85,B 0,C 180,E1 8875.813,E2 8875.813} C_VEL
LIN {X 0,Y 441.864,Z 990.235,A -85,B 0,C 180,E1 8877.124,E2 8877.124} C_VEL
LIN {X 0,Y 437.094,Z 1023,A -85,B 0,C 180,E1 8881.519,E2 8881.519} C_VEL
LIN {X 0,Y 433.293,Z 1049.975,A -85,B 0,C 180,E1 8886.307,E2 8886.307} C_VEL
LIN {X 0,Y 430.586,Z 1069.974,A -85,B 0,C 180,E1 8891.551,E2 8891.551} C_VEL
LIN {X 0,Y 429.072,Z 1084.228,A -85,B 0,C 180,E1 8896.781,E2 8896.781} C_VEL
LIN {X 0,Y 428.497,Z 1093.479,A -85,B 0,C 180,E1 8901.875,E2 8901.875} C_VEL
LIN {X 0,Y 428.324,Z 1097.627,A -85,B 0,C 180,E1 8905.946,E2 8905.946} C_VEL
LIN {X 0,Y 428.355,Z 1099,A -85,B 0,C 180,E1 8910,E2 8910} C_VEL
LIN {X 0,Y 428.305,Z 1097.628,A -85,B 0,C 180,E1 8914.054,E2 8914.054} C_VEL
LIN {X 0,Y 428.593,Z 1092.047,A -85,B 0,C 180,E1 8919.063,E2 8919.063} C_VEL
LIN {X 0,Y 429.28,Z 1081.768,A -85,B 0,C 180,E1 8924.293,E2 8924.293} C_VEL
LIN {X 0,Y 431.172,Z 1064.701,A -85,B 0,C 180,E1 8930.02,E2 8930.02} C_VEL
LIN {X 0,Y 433.759,Z 1046.025,A -85,B 0,C 180,E1 8934.487,E2 8934.487} C_VEL
LIN {X 0,Y 437.556,Z 1019.687,A -85,B 0,C 180,E1 8938.974,E2 8938.974} C_VEL
LIN {X 0,Y 442.334,Z 987.304,A -85,B 0,C 180,E1 8943.205,E2 8943.205} C_VEL
LIN {X 0,Y 447.303,Z 951.55,A -85,B 0,C 180,E1 8946.775,E2 8946.775} C_VEL
LIN {X 0,Y 452.467,Z 909.937,A -85,B 0,C 180,E1 8949.864,E2 8949.864} C_VEL
LIN {X 0,Y 457.316,Z 865.582,A -85,B 0,C 180,E1 8952.223,E2 8952.223} C_VEL
LIN {X 0,Y 461.092,Z 822.682,A -85,B 0,C 180,E1 8953.723,E2 8953.723} C_VEL
LIN {X 0,Y 461.225,Z 805.93,A -85,B 0,C 180,E1 8954.198,E2 8954.198} C_VEL
LIN {X 0,Y 438.087,Z 758.197,A -85,B 0,C 180,E1 8957.785,E2 8957.785} C_VEL
LIN {X 0,Y 427.092,Z 738.282,A -85,B 0,C 180,E1 8959.644,E2 8959.644} C_VEL
LIN {X 0,Y 427.027,Z 737.44,A -85,B 0,C 180,E1 8960.341,E2 8960.341} C_VEL
LIN {X 0,Y 426.989,Z 737.44,A -85,B 0,C 180,E1 8965.433,E2 8965.433} C_VEL
LIN {X 0,Y 427.193,Z 737.44,A -85,B 0,C 180,E1 8972.376,E2 8972.376} C_VEL
LIN {X 0,Y 427.451,Z 737.44,A -85,B 0,C 180,E1 8979.252,E2 8979.252} C_VEL
LIN {X 0,Y 427.515,Z 737.44,A -85,B 0,C 180,E1 8985.643,E2 8985.643} C_VEL
LIN {X 0,Y 427.877,Z 737.44,A -85,B 0,C 180,E1 8992.198,E2 8992.198} C_VEL
LIN {X 0,Y 428.235,Z 737.44,A -85,B 0,C 180,E1 8997.969,E2 8997.969} C_VEL
LIN {X 0,Y 428.104,Z 737.44,A -85,B 0,C 180,E1 9004.05,E2 9004.05} C_VEL
LIN {X 0,Y 427.787,Z 737.44,A -85,B 0,C 180,E1 9010.186,E2 9010.186} C_VEL
LIN {X 0,Y 427.515,Z 737.44,A -85,B 0,C 180,E1 9017.027,E2 9017.027} C_VEL
LIN {X 0,Y 427.356,Z 737.44,A -85,B 0,C 180,E1 9022.928,E2 9022.928} C_VEL
LIN {X 0,Y 427.129,Z 737.44,A -85,B 0,C 180,E1 9029.743,E2 9029.743} C_VEL
LIN {X 0,Y 426.944,Z 737.44,A -85,B 0,C 180,E1 9037.063,E2 9037.063} C_VEL
LIN {X 0,Y 426.961,Z 737.44,A -85,B 0,C 180,E1 9042.344,E2 9042.344} C_VEL
LIN {X 0,Y 427.024,Z 737.44,A -85,B 0,C 180,E1 9048.107,E2 9048.107} C_VEL
LIN {X 0,Y 427.006,Z 737.44,A -85,B 0,C 180,E1 9050.342,E2 9050.342} C_VEL
LIN {X 0,Y 429.339,Z 743.066,A -85,B 0,C 180,E1 9050.802,E2 9050.802} C_VEL
LIN {X 0,Y 446.041,Z 774.106,A -85,B 0,C 180,E1 9053.966,E2 9053.966} C_VEL
LIN {X 0,Y 456.262,Z 797.534,A -85,B 0,C 180,E1 9056.41,E2 9056.41} C_VEL
LIN {X 0,Y 452.044,Z 830.86,A -85,B 0,C 180,E1 9058.555,E2 9058.555} C_VEL
LIN {X 0,Y 446.808,Z 861.792,A -85,B 0,C 180,E1 9061.405,E2 9061.405} C_VEL
LIN {X 0,Y 441.392,Z 888.854,A -85,B 0,C 180,E1 9064.883,E2 9064.883} C_VEL
LIN {X 0,Y 436.522,Z 911.567,A -85,B 0,C 180,E1 9068.91,E2 9068.91} C_VEL
LIN {X 0,Y 432.972,Z 929.131,A -85,B 0,C 180,E1 9073.233,E2 9073.233} C_VEL
LIN {X 0,Y 430.469,Z 943.345,A -85,B 0,C 180,E1 9078.333,E2 9078.333} C_VEL
LIN {X 0,Y 429.384,Z 951.29,A -85,B 0,C 180,E1 9082.911,E2 9082.911} C_VEL
LIN {X 0,Y 429.078,Z 955.455,A -85,B 0,C 180,E1 9087.978,E2 9087.978} C_VEL
LIN {X 0,Y 429.077,Z 955.415,A -85,B 0,C 180,E1 9092.022,E2 9092.022} C_VEL
LIN {X 0,Y 429.433,Z 951.168,A -85,B 0,C 180,E1 9097.088,E2 9097.088} C_VEL
LIN {X 0,Y 430.664,Z 941.982,A -85,B 0,C 180,E1 9102.177,E2 9102.177} C_VEL
LIN {X 0,Y 433.42,Z 927.084,A -85,B 0,C 180,E1 9107.273,E2 9107.273} C_VEL
LIN {X 0,Y 437.451,Z 907.36,A -85,B 0,C 180,E1 9111.842,E2 9111.842} C_VEL
LIN {X 0,Y 442.204,Z 884.825,A -85,B 0,C 180,E1 9115.61,E2 9115.61} C_VEL
LIN {X 0,Y 447.56,Z 857.463,A -85,B 0,C 180,E1 9118.957,E2 9118.957} C_VEL
LIN {X 0,Y 452.722,Z 826.558,A -85,B 0,C 180,E1 9121.671,E2 9121.671} C_VEL
LIN {X 0,Y 456.015,Z 795.528,A -85,B 0,C 180,E1 9123.649,E2 9123.649} C_VEL
LIN {X 0,Y 439.757,Z 761.526,A -85,B 0,C 180,E1 9127.219,E2 9127.219} C_VEL
LIN {X 0,Y 427.052,Z 738.762,A -85,B 0,C 180,E1 9129.506,E2 9129.506} C_VEL
LIN {X 0,Y 426.963,Z 737.44,A -85,B 0,C 180,E1 9129.663,E2 9129.663} C_VEL
LIN {X 0,Y 427.014,Z 737.44,A -85,B 0,C 180,E1 9135.162,E2 9135.162} C_VEL
LIN {X 0,Y 426.996,Z 737.44,A -85,B 0,C 180,E1 9141.265,E2 9141.265} C_VEL
LIN {X 0,Y 427.089,Z 737.44,A -85,B 0,C 180,E1 9148.296,E2 9148.296} C_VEL
LIN {X 0,Y 427.302,Z 737.44,A -85,B 0,C 180,E1 9154.846,E2 9154.846} C_VEL
LIN {X 0,Y 427.576,Z 737.44,A -85,B 0,C 180,E1 9161.424,E2 9161.424} C_VEL
LIN {X 0,Y 427.78,Z 737.44,A -85,B 0,C 180,E1 9167.746,E2 9167.746} C_VEL
LIN {X 0,Y 427.921,Z 737.44,A -85,B 0,C 180,E1 9173.913,E2 9173.913} C_VEL
LIN {X 0,Y 428.222,Z 737.44,A -85,B 0,C 180,E1 9180.005,E2 9180.005} C_VEL
LIN {X 0,Y 427.967,Z 737.44,A -85,B 0,C 180,E1 9186.097,E2 9186.097} C_VEL
LIN {X 0,Y 427.656,Z 737.44,A -85,B 0,C 180,E1 9192.268,E2 9192.268} C_VEL
LIN {X 0,Y 427.468,Z 737.44,A -85,B 0,C 180,E1 9198.592,E2 9198.592} C_VEL
LIN {X 0,Y 427.319,Z 737.44,A -85,B 0,C 180,E1 9205.164,E2 9205.164} C_VEL
LIN {X 0,Y 427.069,Z 737.44,A -85,B 0,C 180,E1 9212.128,E2 9212.128} C_VEL
LIN {X 0,Y 427.023,Z 737.44,A -85,B 0,C 180,E1 9218.739,E2 9218.739} C_VEL
LIN {X 0,Y 427.086,Z 738.048,A -85,B 0,C 180,E1 9220.357,E2 9220.357} C_VEL
LIN {X 0,Y 435.662,Z 753.815,A -85,B 0,C 180,E1 9221.824,E2 9221.824} C_VEL
LIN {X 0,Y 450.848,Z 784.472,A -85,B 0,C 180,E1 9224.258,E2 9224.258} C_VEL
LIN {X 0,Y 461.72,Z 807.169,A -85,B 0,C 180,E1 9225.88,E2 9225.88} C_VEL
LIN {X 0,Y 458.565,Z 851.776,A -85,B 0,C 180,E1 9227.202,E2 9227.202} C_VEL
LIN {X 0,Y 454.011,Z 896.996,A -85,B 0,C 180,E1 9229.361,E2 9229.361} C_VEL
LIN {X 0,Y 448.81,Z 940.255,A -85,B 0,C 180,E1 9232.289,E2 9232.289} C_VEL
LIN {X 0,Y 443.466,Z 979.173,A -85,B 0,C 180,E1 9235.892,E2 9235.892} C_VEL
LIN {X 0,Y 441.864,Z 990.235,A -85,B 0,C 180,E1 9237.124,E2 9237.124} C_VEL
LIN {X 0,Y 436.064,Z 1002.829,A -85,B 0,C 180,E1 9238.544,E2 9238.544} C_VEL
LIN {X 0,Y 430.527,Z 1014.712,A -85,B 0,C 180,E1 9240.075,E2 9240.075} C_VEL
LIN {X 0,Y 426.494,Z 1041.901,A -85,B 0,C 180,E1 9244.61,E2 9244.61} C_VEL
LIN {X 0,Y 423.386,Z 1064.514,A -85,B 0,C 180,E1 9249.595,E2 9249.595} C_VEL
LIN {X 0,Y 421.694,Z 1079.091,A -85,B 0,C 180,E1 9254.379,E2 9254.379} C_VEL
LIN {X 0,Y 420.76,Z 1090.331,A -85,B 0,C 180,E1 9259.635,E2 9259.635} C_VEL
LIN {X 0,Y 420.523,Z 1095.905,A -85,B 0,C 180,E1 9263.799,E2 9263.799} C_VEL
LIN {X 0,Y 420.494,Z 1098.657,A -85,B 0,C 180,E1 9267.936,E2 9267.936} C_VEL
LIN {X 0,Y 420.394,Z 1098.657,A -85,B 0,C 180,E1 9272.064,E2 9272.064} C_VEL
LIN {X 0,Y 420.596,Z 1094.703,A -85,B 0,C 180,E1 9277.238,E2 9277.238} C_VEL
LIN {X 0,Y 421.014,Z 1086.435,A -85,B 0,C 180,E1 9282.46,E2 9282.46} C_VEL
LIN {X 0,Y 422.457,Z 1072.506,A -85,B 0,C 180,E1 9287.989,E2 9287.989} C_VEL
LIN {X 0,Y 424.522,Z 1056.505,A -85,B 0,C 180,E1 9292.35,E2 9292.35} C_VEL
LIN {X 0,Y 428.088,Z 1030.973,A -85,B 0,C 180,E1 9297.372,E2 9297.372} C_VEL
LIN {X 0,Y 432.958,Z 999.164,A -85,B 0,C 180,E1 9302.062,E2 9302.062} C_VEL
LIN {X 0,Y 438.372,Z 962.948,A -85,B 0,C 180,E1 9306.086,E2 9306.086} C_VEL
LIN {X 0,Y 443.786,Z 923.07,A -85,B 0,C 180,E1 9309.408,E2 9309.408} C_VEL
LIN {X 0,Y 449.186,Z 880.009,A -85,B 0,C 180,E1 9312.075,E2 9312.075} C_VEL
LIN {X 0,Y 453.398,Z 839.171,A -85,B 0,C 180,E1 9313.823,E2 9313.823} C_VEL
LIN {X 0,Y 455.072,Z 809.286,A -85,B 0,C 180,E1 9314.714,E2 9314.714} C_VEL
LIN {X 0,Y 433.275,Z 763.435,A -85,B 0,C 180,E1 9318.237,E2 9318.237} C_VEL
LIN {X 0,Y 419.262,Z 738.924,A -85,B 0,C 180,E1 9320.677,E2 9320.677} C_VEL
LIN {X 0,Y 419.127,Z 737.44,A -85,B 0,C 180,E1 9320.824,E2 9320.824} C_VEL
LIN {X 0,Y 419.067,Z 737.44,A -85,B 0,C 180,E1 9327.183,E2 9327.183} C_VEL
LIN {X 0,Y 419.246,Z 737.44,A -85,B 0,C 180,E1 9331.997,E2 9331.997} C_VEL
LIN {X 0,Y 419.514,Z 737.44,A -85,B 0,C 180,E1 9338.841,E2 9338.841} C_VEL
LIN {X 0,Y 419.595,Z 737.44,A -85,B 0,C 180,E1 9345.366,E2 9345.366} C_VEL
LIN {X 0,Y 419.938,Z 737.44,A -85,B 0,C 180,E1 9351.704,E2 9351.704} C_VEL
LIN {X 0,Y 420.321,Z 737.44,A -85,B 0,C 180,E1 9357.931,E2 9357.931} C_VEL
LIN {X 0,Y 420.185,Z 737.44,A -85,B 0,C 180,E1 9364.127,E2 9364.127} C_VEL
LIN {X 0,Y 419.85,Z 737.44,A -85,B 0,C 180,E1 9370.381,E2 9370.381} C_VEL
LIN {X 0,Y 419.661,Z 737.44,A -85,B 0,C 180,E1 9376.768,E2 9376.768} C_VEL
LIN {X 0,Y 419.389,Z 737.44,A -85,B 0,C 180,E1 9383.389,E2 9383.389} C_VEL
LIN {X 0,Y 419.181,Z 737.44,A -85,B 0,C 180,E1 9390.365,E2 9390.365} C_VEL
LIN {X 0,Y 419.038,Z 737.44,A -85,B 0,C 180,E1 9397.358,E2 9397.358} C_VEL
LIN {X 0,Y 418.991,Z 737.44,A -85,B 0,C 180,E1 9403.724,E2 9403.724} C_VEL
LIN {X 0,Y 419.044,Z 737.475,A -85,B 0,C 180,E1 9409.268,E2 9409.268} C_VEL
LIN {X 0,Y 421.424,Z 743.067,A -85,B 0,C 180,E1 9409.736,E2 9409.736} C_VEL
LIN {X 0,Y 438.47,Z 774.181,A -85,B 0,C 180,E1 9413.063,E2 9413.063} C_VEL
LIN {X 0,Y 449.845,Z 801.225,A -85,B 0,C 180,E1 9415.937,E2 9415.937} C_VEL
LIN {X 0,Y 445.017,Z 836.207,A -85,B 0,C 180,E1 9418.303,E2 9418.303} C_VEL
LIN {X 0,Y 439.624,Z 865.784,A -85,B 0,C 180,E1 9421.175,E2 9421.175} C_VEL
LIN {X 0,Y 434.036,Z 892.126,A -85,B 0,C 180,E1 9424.704,E2 9424.704} C_VEL
LIN {X 0,Y 429.045,Z 914.349,A -85,B 0,C 180,E1 9428.796,E2 9428.796} C_VEL
LIN {X 0,Y 425.17,Z 932.397,A -85,B 0,C 180,E1 9433.449,E2 9433.449} C_VEL
LIN {X 0,Y 422.707,Z 945.955,A -85,B 0,C 180,E1 9438.639,E2 9438.639} C_VEL
LIN {X 0,Y 421.591,Z 953.911,A -85,B 0,C 180,E1 9443.815,E2 9443.815} C_VEL
LIN {X 0,Y 421.32,Z 956.808,A -85,B 0,C 180,E1 9447.941,E2 9447.941} C_VEL
LIN {X 0,Y 421.32,Z 956.768,A -85,B 0,C 180,E1 9452.059,E2 9452.059} C_VEL
LIN {X 0,Y 421.706,Z 952.596,A -85,B 0,C 180,E1 9457.219,E2 9457.219} C_VEL
LIN {X 0,Y 423.062,Z 943.481,A -85,B 0,C 180,E1 9462.399,E2 9462.399} C_VEL
LIN {X 0,Y 426.002,Z 928.646,A -85,B 0,C 180,E1 9467.583,E2 9467.583} C_VEL
LIN {X 0,Y 430.282,Z 908.985,A -85,B 0,C 180,E1 9472.225,E2 9472.225} C_VEL
LIN {X 0,Y 435.275,Z 886.538,A -85,B 0,C 180,E1 9476.048,E2 9476.048} C_VEL
LIN {X 0,Y 440.858,Z 859.313,A -85,B 0,C 180,E1 9479.441,E2 9479.441} C_VEL
LIN {X 0,Y 446.302,Z 828.342,A -85,B 0,C 180,E1 9482.208,E2 9482.208} C_VEL
LIN {X 0,Y 450.034,Z 799.629,A -85,B 0,C 180,E1 9484.049,E2 9484.049} C_VEL
LIN {X 0,Y 434.499,Z 766.274,A -85,B 0,C 180,E1 9487.677,E2 9487.677} C_VEL
LIN {X 0,Y 419.087,Z 738.577,A -85,B 0,C 180,E1 9490.601,E2 9490.601} C_VEL
LIN {X 0,Y 419.01,Z 737.44,A -85,B 0,C 180,E1 9490.657,E2 9490.657} C_VEL
LIN {X 0,Y 419.02,Z 737.44,A -85,B 0,C 180,E1 9496.658,E2 9496.658} C_VEL
LIN {X 0,Y 419.047,Z 737.44,A -85,B 0,C 180,E1 9502.641,E2 9502.641} C_VEL
LIN {X 0,Y 419.215,Z 737.44,A -85,B 0,C 180,E1 9510.084,E2 9510.084} C_VEL
LIN {X 0,Y 419.396,Z 737.44,A -85,B 0,C 180,E1 9516.611,E2 9516.611} C_VEL
LIN {X 0,Y 419.744,Z 737.44,A -85,B 0,C 180,E1 9523.236,E2 9523.236} C_VEL
LIN {X 0,Y 419.916,Z 737.44,A -85,B 0,C 180,E1 9529.621,E2 9529.621} C_VEL
LIN {X 0,Y 420.189,Z 737.44,A -85,B 0,C 180,E1 9535.873,E2 9535.873} C_VEL
LIN {X 0,Y 420.324,Z 737.44,A -85,B 0,C 180,E1 9542.069,E2 9542.069} C_VEL
LIN {X 0,Y 419.955,Z 737.44,A -85,B 0,C 180,E1 9548.296,E2 9548.296} C_VEL
LIN {X 0,Y 419.669,Z 737.44,A -85,B 0,C 180,E1 9554.632,E2 9554.632} C_VEL
LIN {X 0,Y 419.476,Z 737.44,A -85,B 0,C 180,E1 9561.161,E2 9561.161} C_VEL
LIN {X 0,Y 419.247,Z 737.44,A -85,B 0,C 180,E1 9568.003,E2 9568.003} C_VEL
LIN {X 0,Y 419.076,Z 737.44,A -85,B 0,C 180,E1 9575.315,E2 9575.315} C_VEL
LIN {X 0,Y 419.147,Z 737.629,A -85,B 0,C 180,E1 9579.282,E2 9579.282} C_VEL
LIN {X 0,Y 421.533,Z 743.069,A -85,B 0,C 180,E1 9579.75,E2 9579.75} C_VEL
LIN {X 0,Y 440.556,Z 777.739,A -85,B 0,C 180,E1 9582.971,E2 9582.971} C_VEL
LIN {X 0,Y 455.242,Z 809.493,A -85,B 0,C 180,E1 9585.309,E2 9585.309} C_VEL
LIN {X 0,Y 451.726,Z 855.583,A -85,B 0,C 180,E1 9586.781,E2 9586.781} C_VEL
LIN {X 0,Y 446.726,Z 900.016,A -85,B 0,C 180,E1 9589.05,E2 9589.05} C_VEL
LIN {X 0,Y 441.077,Z 943.062,A -85,B 0,C 180,E1 9592.138,E2 9592.138} C_VEL
LIN {X 0,Y 435.799,Z 980.078,A -85,B 0,C 180,E1 9595.677,E2 9595.677} C_VEL
LIN {X 0,Y 430.847,Z 1012.698,A -85,B 0,C 180,E1 9599.778,E2 9599.778} C_VEL
LIN {X 0,Y 430.527,Z 1014.712,A -85,B 0,C 180,E1 9600.075,E2 9600.075} C_VEL
LIN {X 0,Y 425.023,Z 1025.977,A -85,B 0,C 180,E1 9601.725,E2 9601.725} C_VEL
LIN {X 0,Y 419.486,Z 1036.491,A -85,B 0,C 180,E1 9603.477,E2 9603.477} C_VEL
LIN {X 0,Y 415.989,Z 1060.69,A -85,B 0,C 180,E1 9608.657,E2 9608.657} C_VEL
LIN {X 0,Y 414.094,Z 1077.607,A -85,B 0,C 180,E1 9613.54,E2 9613.54} C_VEL
LIN {X 0,Y 413.028,Z 1088.406,A -85,B 0,C 180,E1 9618.369,E2 9618.369} C_VEL
LIN {X 0,Y 412.625,Z 1095.905,A -85,B 0,C 180,E1 9623.68,E2 9623.68} C_VEL
LIN {X 0,Y 412.587,Z 1098.657,A -85,B 0,C 180,E1 9627.897,E2 9627.897} C_VEL
LIN {X 0,Y 412.489,Z 1098.657,A -85,B 0,C 180,E1 9632.103,E2 9632.103} C_VEL
LIN {X 0,Y 412.711,Z 1094.094,A -85,B 0,C 180,E1 9637.911,E2 9637.911} C_VEL
LIN {X 0,Y 413.308,Z 1084.924,A -85,B 0,C 180,E1 9643.406,E2 9643.406} C_VEL
LIN {X 0,Y 414.568,Z 1072.858,A -85,B 0,C 180,E1 9648.003,E2 9648.003} C_VEL
LIN {X 0,Y 417.138,Z 1052.72,A -85,B 0,C 180,E1 9653.218,E2 9653.218} C_VEL
LIN {X 0,Y 420.638,Z 1028.788,A -85,B 0,C 180,E1 9657.898,E2 9657.898} C_VEL
LIN {X 0,Y 425.705,Z 996.691,A -85,B 0,C 180,E1 9662.646,E2 9662.646} C_VEL
LIN {X 0,Y 431.237,Z 960.837,A -85,B 0,C 180,E1 9666.644,E2 9666.644} C_VEL
LIN {X 0,Y 437.277,Z 919.326,A -85,B 0,C 180,E1 9670.169,E2 9670.169} C_VEL
LIN {X 0,Y 442.746,Z 878.587,A -85,B 0,C 180,E1 9672.717,E2 9672.717} C_VEL
LIN {X 0,Y 447.279,Z 837.362,A -85,B 0,C 180,E1 9674.484,E2 9674.484} C_VEL
LIN {X 0,Y 448.706,Z 812.323,A -85,B 0,C 180,E1 9675.263,E2 9675.263} C_VEL
LIN {X 0,Y 428.47,Z 768.634,A -85,B 0,C 180,E1 9678.703,E2 9678.703} C_VEL
LIN {X 0,Y 411.324,Z 738.903,A -85,B 0,C 180,E1 9681.806,E2 9681.806} C_VEL
LIN {X 0,Y 411.184,Z 737.44,A -85,B 0,C 180,E1 9681.869,E2 9681.869} C_VEL
LIN {X 0,Y 411.174,Z 737.44,A -85,B 0,C 180,E1 9688.966,E2 9688.966} C_VEL
LIN {X 0,Y 411.361,Z 737.44,A -85,B 0,C 180,E1 9693.787,E2 9693.787} C_VEL
LIN {X 0,Y 411.639,Z 737.44,A -85,B 0,C 180,E1 9700.665,E2 9700.665} C_VEL
LIN {X 0,Y 411.733,Z 737.44,A -85,B 0,C 180,E1 9707.25,E2 9707.25} C_VEL
LIN {X 0,Y 412.137,Z 737.44,A -85,B 0,C 180,E1 9713.668,E2 9713.668} C_VEL
LIN {X 0,Y 412.403,Z 737.44,A -85,B 0,C 180,E1 9719.995,E2 9719.995} C_VEL
LIN {X 0,Y 412.097,Z 737.44,A -85,B 0,C 180,E1 9726.322,E2 9726.322} C_VEL
LIN {X 0,Y 411.825,Z 737.44,A -85,B 0,C 180,E1 9732.736,E2 9732.736} C_VEL
LIN {X 0,Y 411.621,Z 737.44,A -85,B 0,C 180,E1 9739.324,E2 9739.324} C_VEL
LIN {X 0,Y 411.335,Z 737.44,A -85,B 0,C 180,E1 9746.203,E2 9746.203} C_VEL
LIN {X 0,Y 411.167,Z 737.44,A -85,B 0,C 180,E1 9753.517,E2 9753.517} C_VEL
LIN {X 0,Y 411.015,Z 737.44,A -85,B 0,C 180,E1 9759.327,E2 9759.327} C_VEL
LIN {X 0,Y 411.053,Z 737.44,A -85,B 0,C 180,E1 9765.589,E2 9765.589} C_VEL
LIN {X 0,Y 411.206,Z 737.44,A -85,B 0,C 180,E1 9768.113,E2 9768.113} C_VEL
LIN {X 0,Y 413.641,Z 743.169,A -85,B 0,C 180,E1 9768.632,E2 9768.632} C_VEL
LIN {X 0,Y 431.097,Z 774.648,A -85,B 0,C 180,E1 9772.162,E2 9772.162} C_VEL
LIN {X 0,Y 443.55,Z 804.064,A -85,B 0,C 180,E1 9775.41,E2 9775.41} C_VEL
LIN {X 0,Y 438.511,Z 838.146,A -85,B 0,C 180,E1 9777.777,E2 9777.777} C_VEL
LIN {X 0,Y 432.906,Z 867.524,A -85,B 0,C 180,E1 9780.685,E2 9780.685} C_VEL
LIN {X 0,Y 427.054,Z 893.754,A -85,B 0,C 180,E1 9784.26,E2 9784.26} C_VEL
LIN {X 0,Y 421.82,Z 915.902,A -85,B 0,C 180,E1 9788.415,E2 9788.415} C_VEL
LIN {X 0,Y 417.719,Z 933.891,A -85,B 0,C 180,E1 9793.145,E2 9793.145} C_VEL
LIN {X 0,Y 415.076,Z 947.381,A -85,B 0,C 180,E1 9798.427,E2 9798.427} C_VEL
LIN {X 0,Y 413.835,Z 955.293,A -85,B 0,C 180,E1 9803.699,E2 9803.699} C_VEL
LIN {X 0,Y 413.557,Z 958.158,A -85,B 0,C 180,E1 9807.902,E2 9807.902} C_VEL
LIN {X 0,Y 413.558,Z 958.119,A -85,B 0,C 180,E1 9812.098,E2 9812.098} C_VEL
LIN {X 0,Y 413.973,Z 953.992,A -85,B 0,C 180,E1 9817.354,E2 9817.354} C_VEL
LIN {X 0,Y 415.451,Z 944.928,A -85,B 0,C 180,E1 9822.63,E2 9822.63} C_VEL
LIN {X 0,Y 418.561,Z 930.155,A -85,B 0,C 180,E1 9827.906,E2 9827.906} C_VEL
LIN {X 0,Y 423.113,Z 910.568,A -85,B 0,C 180,E1 9832.623,E2 9832.623} C_VEL
LIN {X 0,Y 428.724,Z 886.451,A -85,B 0,C 180,E1 9836.76,E2 9836.76} C_VEL
LIN {X 0,Y 434.621,Z 858.771,A -85,B 0,C 180,E1 9840.194,E2 9840.194} C_VEL
LIN {X 0,Y 440.296,Z 827.542,A -85,B 0,C 180,E1 9842.959,E2 9842.959} C_VEL
LIN {X 0,Y 443.453,Z 802.343,A -85,B 0,C 180,E1 9844.62,E2 9844.62} C_VEL
LIN {X 0,Y 428.189,Z 768.969,A -85,B 0,C 180,E1 9848.372,E2 9848.372} C_VEL
LIN {X 0,Y 412.402,Z 741.918,A -85,B 0,C 180,E1 9851.479,E2 9851.479} C_VEL
LIN {X 0,Y 410.987,Z 737.44,A -85,B 0,C 180,E1 9851.885,E2 9851.885} C_VEL
LIN {X 0,Y 411.047,Z 737.44,A -85,B 0,C 180,E1 9858.484,E2 9858.484} C_VEL
LIN {X 0,Y 411.094,Z 737.44,A -85,B 0,C 180,E1 9864.118,E2 9864.118} C_VEL
LIN {X 0,Y 411.294,Z 737.44,A -85,B 0,C 180,E1 9871.419,E2 9871.419} C_VEL
LIN {X 0,Y 411.549,Z 737.44,A -85,B 0,C 180,E1 9878.423,E2 9878.423} C_VEL
LIN {X 0,Y 411.838,Z 737.44,A -85,B 0,C 180,E1 9885.095,E2 9885.095} C_VEL
LIN {X 0,Y 412.083,Z 737.44,A -85,B 0,C 180,E1 9891.555,E2 9891.555} C_VEL
LIN {X 0,Y 412.275,Z 737.44,A -85,B 0,C 180,E1 9897.901,E2 9897.901} C_VEL
LIN {X 0,Y 412.157,Z 737.44,A -85,B 0,C 180,E1 9904.218,E2 9904.218} C_VEL
LIN {X 0,Y 411.881,Z 737.44,A -85,B 0,C 180,E1 9910.595,E2 9910.595} C_VEL
LIN {X 0,Y 411.654,Z 737.44,A -85,B 0,C 180,E1 9917.115,E2 9917.115} C_VEL
LIN {X 0,Y 411.45,Z 737.44,A -85,B 0,C 180,E1 9923.88,E2 9923.88} C_VEL
LIN {X 0,Y 411.314,Z 737.44,A -85,B 0,C 180,E1 9928.592,E2 9928.592} C_VEL
LIN {X 0,Y 411.14,Z 737.44,A -85,B 0,C 180,E1 9936.103,E2 9936.103} C_VEL
LIN {X 0,Y 411.204,Z 737.44,A -85,B 0,C 180,E1 9938.13,E2 9938.13} C_VEL
LIN {X 0,Y 413.752,Z 743.219,A -85,B 0,C 180,E1 9938.673,E2 9938.673} C_VEL
LIN {X 0,Y 434.021,Z 779.415,A -85,B 0,C 180,E1 9942.247,E2 9942.247} C_VEL
LIN {X 0,Y 448.975,Z 812.718,A -85,B 0,C 180,E1 9944.78,E2 9944.78} C_VEL
LIN {X 0,Y 445.188,Z 856.583,A -85,B 0,C 180,E1 9946.235,E2 9946.235} C_VEL
LIN {X 0,Y 440.214,Z 898.149,A -85,B 0,C 180,E1 9948.395,E2 9948.395} C_VEL
LIN {X 0,Y 434.314,Z 939.713,A -85,B 0,C 180,E1 9951.442,E2 9951.442} C_VEL
LIN {X 0,Y 428.521,Z 978.305,A -85,B 0,C 180,E1 9955.167,E2 9955.167} C_VEL
LIN {X 0,Y 423.466,Z 1010.709,A -85,B 0,C 180,E1 9959.261,E2 9959.261} C_VEL
LIN {X 0,Y 419.486,Z 1036.491,A -85,B 0,C 180,E1 9963.477,E2 9963.477} C_VEL
LIN {X 0,Y 414.059,Z 1046.337,A -85,B 0,C 180,E1 9965.331,E2 9965.331} C_VEL
LIN {X 0,Y 408.924,Z 1055.24,A -85,B 0,C 180,E1 9967.316,E2 9967.316} C_VEL
LIN {X 0,Y 406.522,Z 1074.461,A -85,B 0,C 180,E1 9972.666,E2 9972.666} C_VEL
LIN {X 0,Y 405.158,Z 1088.195,A -85,B 0,C 180,E1 9978.14,E2 9978.14} C_VEL
LIN {X 0,Y 404.748,Z 1095.905,A -85,B 0,C 180,E1 9983.557,E2 9983.557} C_VEL
LIN {X 0,Y 404.688,Z 1098.657,A -85,B 0,C 180,E1 9987.856,E2 9987.856} C_VEL
LIN {X 0,Y 404.599,Z 1098.657,A -85,B 0,C 180,E1 9992.144,E2 9992.144} C_VEL
LIN {X 0,Y 404.792,Z 1094.406,A -85,B 0,C 180,E1 9997.788,E2 9997.788} C_VEL
LIN {X 0,Y 405.323,Z 1085.998,A -85,B 0,C 180,E1 10002.951,E2 10002.951} C_VEL
LIN {X 0,Y 406.981,Z 1070.146,A -85,B 0,C 180,E1 10008.698,E2 10008.698} C_VEL
LIN {X 0,Y 409.65,Z 1049.463,A -85,B 0,C 180,E1 10013.987,E2 10013.987} C_VEL
LIN {X 0,Y 413.467,Z 1024.876,A -85,B 0,C 180,E1 10018.724,E2 10018.724} C_VEL
LIN {X 0,Y 418.322,Z 994.961,A -85,B 0,C 180,E1 10023.142,E2 10023.142} C_VEL
LIN {X 0,Y 424.51,Z 956.194,A -85,B 0,C 180,E1 10027.509,E2 10027.509} C_VEL
LIN {X 0,Y 430.662,Z 917.498,A -85,B 0,C 180,E1 10030.841,E2 10030.841} C_VEL
LIN {X 0,Y 436.446,Z 876.785,A -85,B 0,C 180,E1 10033.407,E2 10033.407} C_VEL
LIN {X 0,Y 441.218,Z 835.718,A -85,B 0,C 180,E1 10035.164,E2 10035.164} C_VEL
LIN {X 0,Y 442.466,Z 815.57,A -85,B 0,C 180,E1 10035.808,E2 10035.808} C_VEL
LIN {X 0,Y 423.863,Z 774.113,A -85,B 0,C 180,E1 10039.152,E2 10039.152} C_VEL
LIN {X 0,Y 405.193,Z 742.613,A -85,B 0,C 180,E1 10042.622,E2 10042.622} C_VEL
LIN {X 0,Y 403.284,Z 737.44,A -85,B 0,C 180,E1 10043.079,E2 10043.079} C_VEL
LIN {X 0,Y 403.306,Z 737.44,A -85,B 0,C 180,E1 10050.786,E2 10050.786} C_VEL
LIN {X 0,Y 403.609,Z 737.44,A -85,B 0,C 180,E1 10057.965,E2 10057.965} C_VEL
LIN {X 0,Y 403.726,Z 737.44,A -85,B 0,C 180,E1 10064.777,E2 10064.777} C_VEL
LIN {X 0,Y 404.082,Z 737.44,A -85,B 0,C 180,E1 10071.376,E2 10071.376} C_VEL
LIN {X 0,Y 404.512,Z 737.44,A -85,B 0,C 180,E1 10077.85,E2 10077.85} C_VEL
LIN {X 0,Y 404.347,Z 737.44,A -85,B 0,C 180,E1 10084.289,E2 10084.289} C_VEL
LIN {X 0,Y 403.978,Z 737.44,A -85,B 0,C 180,E1 10090.794,E2 10090.794} C_VEL
LIN {X 0,Y 403.756,Z 737.44,A -85,B 0,C 180,E1 10097.449,E2 10097.449} C_VEL
LIN {X 0,Y 403.449,Z 737.44,A -85,B 0,C 180,E1 10104.372,E2 10104.372} C_VEL
LIN {X 0,Y 403.254,Z 737.44,A -85,B 0,C 180,E1 10111.701,E2 10111.701} C_VEL
LIN {X 0,Y 403.05,Z 737.44,A -85,B 0,C 180,E1 10117.924,E2 10117.924} C_VEL
LIN {X 0,Y 403.138,Z 737.44,A -85,B 0,C 180,E1 10124.476,E2 10124.476} C_VEL
LIN {X 0,Y 403.187,Z 737.907,A -85,B 0,C 180,E1 10126.91,E2 10126.91} C_VEL
LIN {X 0,Y 405.867,Z 743.323,A -85,B 0,C 180,E1 10127.466,E2 10127.466} C_VEL
LIN {X 0,Y 423.65,Z 774.987,A -85,B 0,C 180,E1 10131.201,E2 10131.201} C_VEL
LIN {X 0,Y 437.144,Z 807.421,A -85,B 0,C 180,E1 10134.908,E2 10134.908} C_VEL
LIN {X 0,Y 431.859,Z 841.05,A -85,B 0,C 180,E1 10137.321,E2 10137.321} C_VEL
LIN {X 0,Y 426.199,Z 869.24,A -85,B 0,C 180,E1 10140.177,E2 10140.177} C_VEL
LIN {X 0,Y 420.102,Z 895.351,A -85,B 0,C 180,E1 10143.802,E2 10143.802} C_VEL
LIN {X 0,Y 414.59,Z 917.427,A -85,B 0,C 180,E1 10148.019,E2 10148.019} C_VEL
LIN {X 0,Y 410.258,Z 935.363,A -85,B 0,C 180,E1 10152.829,E2 10152.829} C_VEL
LIN {X 0,Y 407.437,Z 948.789,A -85,B 0,C 180,E1 10158.207,E2 10158.207} C_VEL
LIN {X 0,Y 406.103,Z 956.661,A -85,B 0,C 180,E1 10163.579,E2 10163.579} C_VEL
LIN {X 0,Y 405.793,Z 959.507,A -85,B 0,C 180,E1 10167.862,E2 10167.862} C_VEL
LIN {X 0,Y 405.793,Z 959.469,A -85,B 0,C 180,E1 10172.138,E2 10172.138} C_VEL
LIN {X 0,Y 406.258,Z 955.371,A -85,B 0,C 180,E1 10177.495,E2 10177.495} C_VEL
LIN {X 0,Y 407.836,Z 946.353,A -85,B 0,C 180,E1 10182.87,E2 10182.87} C_VEL
LIN {X 0,Y 411.146,Z 931.627,A -85,B 0,C 180,E1 10188.24,E2 10188.24} C_VEL
LIN {X 0,Y 415.964,Z 912.12,A -85,B 0,C 180,E1 10193.034,E2 10193.034} C_VEL
LIN {X 0,Y 421.832,Z 888.091,A -85,B 0,C 180,E1 10197.233,E2 10197.233} C_VEL
LIN {X 0,Y 427.999,Z 860.542,A -85,B 0,C 180,E1 10200.711,E2 10200.711} C_VEL
LIN {X 0,Y 433.928,Z 829.404,A -85,B 0,C 180,E1 10203.519,E2 10203.519} C_VEL
LIN {X 0,Y 437.071,Z 805.503,A -85,B 0,C 180,E1 10205.152,E2 10205.152} C_VEL
